	//----------------------------------------------------------------------------------------------
	// Execution of torquelimiting functionality
	//----------------------------------------------------------------------------------------------
	REGION EXECUTION_OF_TORQUELIMTING
	  // Statemachine for torquelimiting 
	  REPEAT
	    #tempStateChangeActive := FALSE;
	    CASE #statTorqueLimitingState OF
	      #NO_TORQUE_LIMITING_ACTIVE:
	        ; // Torquelimiting disable
	        // #instTorqueLimiting(Axis := #axis, V01.00.03 Dont Call MC_TORQUELIMITING if disabled
	        //                     Enable := FALSE);
	        
	      #TORQUE_LIMITING_DISABLE:
	        // Torquelimiting disable
	        #instTorqueLimiting(Axis := #axis,
	                            Enable := FALSE);
	        
	        // Check state of torque limting
	        IF (#instTorqueLimiting.Busy = FALSE)
	        THEN
	          // set next state
	          #statTorqueLimitingState := #NO_TORQUE_LIMITING_ACTIVE;
	        ELSE
	          ; // Waiting for MC_Torquelimiting is not busy
	        END_IF;
	        
	      #TORQUE_LIMTING_SELECTED:
	        // No extended homing function active
	        #instTorqueLimiting(Axis := #axis,
	                            Enable := #statExtendedCommand.%X1,
	                            Limit := #configuration.torqueLimiting.limit,
	                            Mode := #configuration.torqueLimiting.mode);
	        
	        IF (#instTorqueLimiting.Busy = FALSE) THEN
	          // Reset state
	          #statTorqueLimitingState := #NO_TORQUE_LIMITING_ACTIVE;
	        END_IF;
	        
	        (*
	        V1.00.03 Not required anymore
	      #AUTOMATIC_MODE_CHANGE:
	        // In this state the torquelimiting function is operating with Mode 1 (Fixed stop detection) until inClamping = FALSE
	        #instTorqueLimiting(Axis := #axis,
	                            Enable := TRUE,
	                            Limit := #configuration.homing.extendedModeTorqueLimit); // V01.00.03 Always use configured value
	        
	        IF (#configuration.torqueLimiting.mode = #MODE_FIXED_STOP_DETECTION)
	          OR (#instTorqueLimiting.InClamping = FALSE)
	        THEN
	          // Change state
	          #statTorqueLimitingState := #TORQUE_LIMTING_SELECTED;
	          #tempStateChangeActive := TRUE;
	        ELSE
	          ; // Wait for InClamping = FALSE
	        END_IF;
	        *)
	        
	      #FIXED_STOP_DETECTION_ACTIVE:
	        // Extended homing function active
	        #instTorqueLimiting(Axis := #axis,
	                            Enable := TRUE,
	                            Limit := #configuration.homing.extendedModeTorqueLimit, // V01.00.03 Always use configured value
	                            Mode := #MODE_FIXED_STOP_DETECTION);
	        
	        IF ((#statHomingSubState = #HOMING_IDLE) AND (#statBasicMotionState = #ACTIVE_HOMING_SELECTED))
	        THEN
	          // Fixed stop process has finished - Axis is still in clamping
	          #statTorqueLimitingState := #FIXED_STOP_DETECTION_FINISHED;
	          #tempStateChangeActive := TRUE;
	          
	        ELSIF (#statBasicMotionState <> #ACTIVE_HOMING_SELECTED)
	        THEN
	          // Error occurred - change state depending on inClamping
	          IF (#instTorqueLimiting.InClamping = TRUE)
	          THEN
	            // Axis is in clamping
	            #statTorqueLimitingState := #FIXED_STOP_DETECTION_ERROR_IN_CLAMPING;
	            #tempStateChangeActive := TRUE;
	          ELSE
	            // Axis is in not clamping
	            #statTorqueLimitingState := #FIXED_STOP_DETECTION_ERROR_NOT_IN_CLAMPING;
	            #tempStateChangeActive := TRUE;
	          END_IF;
	          
	        ELSE
	          ; // Fixed stop detection is running
	        END_IF;
	        
	      #FIXED_STOP_DETECTION_FINISHED:
	        // Homing on fixed stop process has finished
	        #instTorqueLimiting(Axis := #axis,
	                            Enable := TRUE,
	                            Limit := #configuration.homing.extendedModeTorqueLimit, // V01.00.03 Always use configured value
	                            Mode := #MODE_FIXED_STOP_DETECTION);
	        
	        IF (#instTorqueLimiting.InClamping = FALSE)
	        THEN
	          // InClamping = FALSE
	          IF (#statExtendedCommand.%X1 = TRUE) // Torquelimiting
	          THEN
	            #statTorqueLimitingState := #TORQUE_LIMTING_SELECTED;
	          ELSE
	            #statTorqueLimitingState := #TORQUE_LIMITING_DISABLE;
	          END_IF;
	          #tempStateChangeActive := TRUE;
	        ELSE
	          // InClamping = TRUE
	          IF (#statExtendedCommand.%X1 = TRUE) // Torquelimiting
	            AND (#configuration.torqueLimiting.mode = #MODE_FIXED_STOP_DETECTION)
	          THEN
	            // Change State
	            #statTorqueLimitingState := #TORQUE_LIMTING_SELECTED;
	            #tempStateChangeActive := TRUE;
	          ELSE
	            ; // Wait for inClamping = FALSE
	          END_IF;
	        END_IF;
	        
	      #FIXED_STOP_DETECTION_ERROR_IN_CLAMPING:
	        // Errorstate, torquelimiting is still active and axis not in clamping
	        #instTorqueLimiting(Axis := #axis,
	                            Enable := TRUE,
	                            Limit := #configuration.homing.extendedModeTorqueLimit, // V01.00.03 Always use configured value
	                            Mode := #MODE_FIXED_STOP_DETECTION);
	        
	        IF (#instTorqueLimiting.InClamping = FALSE)
	        THEN
	          // InClamping = FALSE -> reset torque limiting state
	          #statTorqueLimitingState := #TORQUE_LIMITING_DISABLE;
	          // Torquelimiting disable
	          #tempStateChangeActive := TRUE;
	        END_IF;
	        
	      #FIXED_STOP_DETECTION_ERROR_NOT_IN_CLAMPING:
	        // Errorstate, torquelimiting is still active and axis in clamping
	        #instTorqueLimiting(Axis := #axis,
	                            Enable := TRUE,
	                            Limit := #configuration.homing.extendedModeTorqueLimit, // V01.00.03 Always use configured value
	                            Mode := #MODE_FIXED_STOP_DETECTION);
	        
	        IF (#instTorqueLimiting.InClamping = TRUE)
	        THEN
	          // InClamping = TRUE -> change state
	          #statTorqueLimitingState := #FIXED_STOP_DETECTION_ERROR_IN_CLAMPING;
	          #tempStateChangeActive := TRUE;
	          
	        ELSIF (#statBasicMotionState <> #NO_SELECTION)
	          OR (#statSupImpMotionState <> #NO_SELECTION)
	          OR (#statPassiveHomingState <> #NO_HOMING_ACTIVE)
	        THEN
	          // New valid command is set -> reset error state
	          #statTorqueLimitingState := #TORQUE_LIMITING_DISABLE;
	          #tempStateChangeActive := TRUE;
	          
	        ELSE
	          ; // Waiting for new command or axis is getting in clamping
	        END_IF;
	      ELSE
	        // Errorhandling
	        #statStatus := #ERR_UNDEFINED_TORQUE_LIMITING_STATE;
	        #statErrorUserCleared := TRUE;
	        #diagnostics.basicMotionState := #statBasicMotionState;
	        #diagnostics.superimposedMotionState := #statSupImpMotionState;
	        #diagnostics.subfunctionStatus := 0;
	        // Set errorstate
	        #statFBState := #FB_ERROR;
	    END_CASE;
	  UNTIL (#tempStateChangeActive = FALSE)
	  END_REPEAT;
	  // Evaluate MC_Command
	  IF (#instTorqueLimiting.Error = TRUE) AND ((#statTorqueLimitingErrorOld = FALSE) OR (#statStatus = #STATUS_SUBSEQUENT_CALL)) THEN
	    // Errorhandling
	    #statStatus := #ERR_MC_TORQUELIMITING;
	    #statErrorAutoCleared := TRUE;
	    #diagnostics.basicMotionState := #statBasicMotionState;
	    #diagnostics.superimposedMotionState := #statSupImpMotionState;
	    #diagnostics.subfunctionStatus := #instTorqueLimiting.ErrorId;
	    #statFBState := #AXIS_STOP_ON_ERROR_SELECTION;
	    
	  ELSIF (#instTorqueLimiting.Error = FALSE) AND ((#statTorqueLimitingErrorOld = TRUE) AND (#statStatus = #ERR_MC_TORQUELIMITING)) THEN
	    #statStatus := #STATUS_SUBSEQUENT_CALL;
	    #statErrorAutoCleared := FALSE;
	  ELSE
	    ;
	  END_IF;
	  
	  #statTorqueLimitingErrorOld := #instTorqueLimiting.Error;
	END_REGION
	
	//----------------------------------------------------------------------------------------------
	// Selection of StopOnError / implementation of fastStop
	//----------------------------------------------------------------------------------------------
	REGION STOP_ON_ERROR
	  // Check for stopping if error occurred during execution of motion commands
	  IF (#statFBState = #AXIS_STOP_ON_ERROR_SELECTION)
	  THEN
	    #statBasicMotionState := #NO_SELECTION;
	    #statSupImpMotionState := #NO_SELECTION;
	    #statPassiveHomingState := #NO_HOMING_ACTIVE;
	    
	    IF (#configuration.generalSettings.stopOnError = TRUE)
	    THEN
	      // Read Statusword only when not already read out
	      IF (#tempStatusWord = 16#0)
	      THEN
	        #tempStatusWord := #axis.StatusWord;
	      END_IF;
	      // Evaluate error
	      IF #tempStatusWord.%X0 THEN
	        ; // Axis enabled
	        IF (#tempStatusWord.%X1 = TRUE) THEN
	          ;// TO Alarm present
	          #statFBState := #AXIS_MOTION;
	        ELSE
	          // No TO alarm present, set fastStop
	          #statBasicMotionState := #FAST_STOP_SELECTED;
	          #statFirstCycleBasicMotion := TRUE;
	          #statFBState := #AXIS_STOP_ON_ERROR_EXECUTION;
	        END_IF;
	        
	      ELSE
	        ; // Axis disabled
	        #statFBState := #AXIS_MOTION;
	      END_IF;
	      
	    ELSE
	      // Dont StopOnError
	      #statFBState := #AXIS_MOTION;
	    END_IF;
	  END_IF;
	  
	  // Implementation of fastStop
	  IF (#statBasicMotionState = #FAST_STOP_SELECTED) THEN
	    // Additional feature: Load emergency stop dynamics (TO) if no valid dynamics are configured for fastStop
	    REGION FASTSTOP SELECTED
	      // Firstcycle of command
	      IF (#statFirstCycleBasicMotion = TRUE) THEN
	        // Reset HALT command
	        #instHalt(Axis := #axis,
	                  Execute := FALSE);
	        #statFirstCycleDone := TRUE;
	        // Check dynamics for fastStop
	        // Load TO emergency Stop dynamics if value <=0 for deceleration is configured
	        IF (#configuration.fastStop.deceleration <= 0) // V1.0.2 Read TO emergencyStop deceleration only if fastStop.deceleration <= 0
	        THEN
	          // Invalid fastStop dynamics configured - read emergency stop dynamics from TO
	          #statDeceleration := #axis.DynamicDefaults.EmergencyDeceleration;
	        ELSE
	          // Valid fastStop dynamics configured
	          #statDeceleration := #configuration.fastStop.deceleration;
	        END_IF;
	        #statJerk := #configuration.fastStop.jerk; // V1.0.2 Use always configuration for jerk value
	        #statAbortAcceleration := #configuration.fastStop.abortAcceleration; // V1.0.2 Use always configuration
	      END_IF;
	      
	      // Call of MC_Command
	      #instHalt(Axis := #axis,
	                Execute := (#statBasicCommand.%X0 OR #statFirstCycleBasicMotion),
	                Deceleration := #statDeceleration,
	                AbortAcceleration := #statAbortAcceleration,
	                Jerk := #statJerk);
	      
	      // Evaluate MC_Command
	      IF (#instHalt.Busy = FALSE) AND
	        (#instHalt.Error = FALSE) AND
	        (#instHalt.Done = FALSE) AND
	        (#instHalt.CommandAborted = FALSE)
	      THEN
	        // Return to NO_SELECTION if command finished
	        #statFBState := #AXIS_MOTION;
	        #statBasicMotionState := #NO_SELECTION;
	        
	      ELSIF (#instHalt.Done = TRUE)
	      THEN
	        IF (#statFirstCycleDone = TRUE)
	        THEN
	          // Command is reset
	          IF (#instTorqueLimiting.Error = FALSE) // V1.00.03 Dont reset error is pending
	          THEN
	            // Reset status not if torquelimiting error is pending
	            #statStatus := #STATUS_SUBSEQUENT_CALL;
	            #statErrorAutoCleared := FALSE;
	          END_IF;
	          
	          #statFirstCycleDone := FALSE;
	        END_IF;
	        
	      ELSIF (#instHalt.Error = TRUE)
	      THEN
	        // Errorhandling
	        #statStatus := #ERR_MC_HALT;
	        #statErrorAutoCleared := TRUE;
	        #diagnostics := #statDiagnostics;
	        #diagnostics.basicMotionState := #statBasicMotionState;
	        #diagnostics.superimposedMotionState := #statSupImpMotionState;
	        #diagnostics.subfunctionStatus := #instHalt.ErrorId;
	        
	      ELSE
	        ; // Command selected
	      END_IF;
	      
	      // Write MC_Command outputs to internal variable
	      #statExeOfBasicMotion := 0;
	      #statExeOfBasicMotion.%X0 := #instHalt.Busy;
	      #statExeOfBasicMotion.%X1 := #instHalt.Done;
	      #statExeOfBasicMotion.%X2 := #instHalt.CommandAborted;
	      #statExeOfBasicMotion.%X3 := #instHalt.Error;
	    END_REGION
	  END_IF;
	END_REGION
	//----------------------------------------------------------------------------------------------
	// Store values and reset variables
	//----------------------------------------------------------------------------------------------
	REGION STORE_AND_RESET
	  // Reset variables to determine first cycle of a new command
	  IF (#statFirstCycleReset = TRUE) THEN
	    #statFirstCycleReset := FALSE;
	  END_IF;
	  IF (#statFirstCycleHoming = TRUE) THEN
	    #statFirstCycleHoming := FALSE;
	  END_IF;
	  #statHomingOld := #tempHoming;
	  
	  IF (#statFirstCycleBasicMotion = TRUE) THEN
	    #statFirstCycleBasicMotion := FALSE;
	  END_IF;
	  #statBasicCommandOld := #statBasicCommand;
	  
	  IF (#statFirstCycleSupImpMotion = TRUE) THEN
	    #statFirstCycleSupImpMotion := FALSE;
	  END_IF;
	  #statSupImpCommandOld := #statSupImpCommand;
	  
	  // Store last values for edge detection
	  #statEnableOld := #enable;
	  #statEnableAxisOld := #enableAxis;
	  #statExtendedCommandOld := #statExtendedCommand;
	  #statPowerErrorOld := #instPower.Error;
	END_REGION
	
	//----------------------------------------------------------------------------------------------
	// Writing outputs
	//----------------------------------------------------------------------------------------------
	REGION WRITING_OF_OUTPUTS
	  // Writing status outputs
	  #resetActive := (#statResetState = #CMD_BUSY);
	  
	  IF (#statErrorUserCleared = TRUE) THEN
	    ; // Reset variables at ErrorUserCleared
	    #statBasicMotionState := #NO_SELECTION;
	    #statExeOfBasicMotion := #NO_SELECTION;
	    #statSupImpMotionState := #NO_SELECTION;
	    #statExeOfSupImpMotionState := #NO_SELECTION;
	    #statExeOfHoming := #NO_SELECTION;
	  END_IF;
	  IF (#instPower.Status = TRUE)
	  THEN
	    // Axis enabled
	    #axisEnabled := TRUE;
	    
	  ELSIF (#instPower.Error = TRUE) AND (#instPower.Status = FALSE)
	  THEN
	    // Reset status if error occurred
	    #axisEnabled := FALSE;
	    
	  ELSIF (#instPower.Busy = FALSE)
	  THEN
	    // Reset if MC_Power is not busy
	    #axisEnabled := FALSE;
	  ELSE
	    ;
	  END_IF;
	  
	  REGION WRITING_BASICMOTION_OUTPUTS
	    // Writing Busy, Done and Aborted outputs for basic motion commands
	    IF (#statBasicMotionState > #NO_SELECTION) AND (#statBasicMotionState < #ACTIVE_HOMING_SELECTED)
	    THEN
	      #commandBusy := #statExeOfBasicMotion.%X0;
	      #commandDone := #statExeOfBasicMotion.%X1;
	      #commandAborted := #statExeOfBasicMotion.%X2;
	      #inVelocity := #statExeOfBasicMotion.%X4;
	    ELSE
	      #commandBusy := FALSE;
	      #commandDone := FALSE;
	      #commandAborted := FALSE;
	      #inVelocity := FALSE;
	    END_IF;
	    
	    // Writing outputs up to LAxisCtrl_SpeedAxis
	    IF (#statTorqueLimitingState = #TORQUE_LIMTING_SELECTED)
	      // OR (#statTorqueLimitingState = #AUTOMATIC_MODE_CHANGE) V1.0.3 TorqueLimtinig = TRUE, only when respective value used 
	    THEN
	      #torqueLimitingSelected := TRUE;
	    ELSE
	      #torqueLimitingSelected := FALSE;
	    END_IF;
	    
	    #inLimitation := #instTorqueLimiting.InLimitation;
	    #fastStopSelected := #statBasicMotionState.%X0;
	    #stopSelected := #statBasicMotionState.%X1;
	    #jogSelected := #statBasicMotionState.%X2 OR #statBasicMotionState.%X3;
	    #moveVelocitySelected := #statBasicMotionState.%X4;
	    // Writing outputs up to LAxisCtrl_PosAxis
	    #inClamping := #instTorqueLimiting.InClamping;
	    #posRelativeSelected := #statBasicMotionState.%X5;
	    #posAbsoluteSelected := #statBasicMotionState.%X6;
	  END_REGION
	  REGION WRITING_HOMING_OUTPUTS
	    // Writing Busy, Done and Aborted outputs for homing
	    IF (#statPassiveHomingState = #STANDARD_HOMING)
	    THEN
	      #homingSelected := TRUE;
	      #homingCommandBusy := #statExeOfHoming.%X0;
	      #homingCommandDone := #statExeOfHoming.%X1;
	      #homingCommandAborted := #statExeOfHoming.%X2;
	    ELSE
	      IF (#statBasicMotionState = #ACTIVE_HOMING_SELECTED)
	      THEN
	        #homingSelected := TRUE;
	        #homingCommandBusy := #statExeOfBasicMotion.%X0;
	        #homingCommandDone := #statExeOfBasicMotion.%X1;
	        #homingCommandAborted := #statExeOfBasicMotion.%X2;
	      ELSE
	        #homingSelected := FALSE;
	        #homingCommandBusy := FALSE;
	        #homingCommandDone := FALSE;
	        #homingCommandAborted := FALSE;
	      END_IF;
	    END_IF;
	  END_REGION
	  REGION WRITING_SUPERIMPOSED_OUTPUTS
	    // Writing outputs for superimposed motion commands
	    IF (#statSupImpMotionState <> #NO_SELECTION)
	    THEN
	      #superimposedBusy := #statExeOfSupImpMotionState.%X0;
	      #superimposedDone := #statExeOfSupImpMotionState.%X1;
	      #superimposedAborted := #statExeOfSupImpMotionState.%X2;
	    ELSE
	      #superimposedBusy := FALSE;
	      #superimposedDone := FALSE;
	      #superimposedAborted := FALSE;
	    END_IF;
	    #posSuperimposedSelected := #statSupImpMotionState.%X0;
	  END_REGION
	END_REGION
	
	//----------------------------------------------------------------------------------------------
	// Error handling 
	//----------------------------------------------------------------------------------------------
	REGION ERROR_HANDLING
	  IF #statErrorUserCleared THEN
	    #valid := FALSE;
	    #busy := TRUE;
	    #error := TRUE;
	    #status := #statStatus;
	    #diagnostics.status := #statStatus;
	    
	  ELSIF #statErrorAutoCleared THEN
	    #valid := FALSE;
	    #busy := TRUE;
	    #error := TRUE;
	    #status := #statStatus;
	    #diagnostics.status := #statStatus;
	    
	  ELSE
	    // Process normal output values
	    #valid := TRUE;
	    #error := FALSE;
	    #status := #statStatus;
	  END_IF;
	END_REGION
END_FUNCTION_BLOCK

FUNCTION_BLOCK "FB_Axis"   // FB30140, LAD
{ S7_Optimized_Access := 'TRUE' }
// stored: AutoNumber false, MemoryReserve 100, SetENOAutomatically false
   VAR_INPUT
      TO_PosAxis : TO_PositioningAxis;
      I_bMan_Enable : Bool;
      I_iHomeMode : Int;
      I_iHomePos : LReal;
   END_VAR
   VAR_IN_OUT
      Ds_Axis : "sAxis";
   END_VAR
   VAR
      instAxis01 { ExternalAccessible := 'False'; ExternalVisible := 'False'; ExternalWritable := 'False'} : "LAxisCtrl_PosAxis";
      instShearAxisStatus { S7_SetPoint := 'True'} : "LAxisCtrl_GetAxisStatusWord";
      RT_Reset { S7_SetPoint := 'True'} : R_TRIG;
      RT_PB { ExternalAccessible := 'False'; ExternalVisible := 'False'; ExternalWritable := 'False'} : Array[0..19] of R_TRIG;   // Störungen / Alarms
      FT_PB { ExternalAccessible := 'False'; ExternalVisible := 'False'; ExternalWritable := 'False'; S7_SetPoint := 'True'} : Array[0..19] of F_TRIG;   // Störungen unterdrücken, Belegung identisch mit "Alarm" / Hide Alarms, identical with "Alarm"
      TON_PB { ExternalAccessible := 'False'; ExternalVisible := 'False'; ExternalWritable := 'False'} : Array[0..19] of TON_TIME;   // Fallende Flanke / Falling edge
      TOF_PB { ExternalAccessible := 'False'; ExternalVisible := 'False'; ExternalWritable := 'False'} : Array[0..19] of TOF_TIME;   // Negativer Impuls / Negative pulse
      i { S7_SetPoint := 'True'} : Int;
      temp_cmd_bEnableAxis { ExternalAccessible := 'False'; ExternalVisible := 'False'; ExternalWritable := 'False'} : Bool;
      temp_cmd_bresetAxis { ExternalAccessible := 'False'; ExternalVisible := 'False'; ExternalWritable := 'False'} : Bool;
      temp_cmd_bjogForward { ExternalAccessible := 'False'; ExternalVisible := 'False'; ExternalWritable := 'False'} : Bool;
      temp_cmd_bjogBackward { ExternalAccessible := 'False'; ExternalVisible := 'False'; ExternalWritable := 'False'} : Bool;
      temp_cmd_bmoveVelocity { ExternalAccessible := 'False'; ExternalVisible := 'False'; ExternalWritable := 'False'} : Bool;
      temp_cmd_bstop { ExternalAccessible := 'False'; ExternalVisible := 'False'; ExternalWritable := 'False'} : Bool;
      temp_cmd_bfastStop { ExternalAccessible := 'False'; ExternalVisible := 'False'; ExternalWritable := 'False'} : Bool;
      temp_cmd_bhoming { ExternalAccessible := 'False'; ExternalVisible := 'False'; ExternalWritable := 'False'} : Bool;
      temp_cmd_bGoToPos { ExternalAccessible := 'False'; ExternalVisible := 'False'; ExternalWritable := 'False'} : Array[0..16] of Bool;
      temp_cmd_iGoToPos : Word;
      temp_cmd_bCallAbsPos : Bool;
      temp_cmd_bRelPos : Bool;
      temp_Para_rJog_Speed { ExternalAccessible := 'False'; ExternalVisible := 'False'; ExternalWritable := 'False'} : LReal;
      temp_cmd_bGoToPosAll { ExternalAccessible := 'False'; ExternalVisible := 'False'; ExternalWritable := 'False'} : Bool;
      temp_configuration { ExternalAccessible := 'False'; ExternalVisible := 'False'; ExternalWritable := 'False'} : "LAxisCtrl_typeAxisConfig";   // Diagnostics structure
      temp_Status { ExternalAccessible := 'False'; ExternalVisible := 'False'; ExternalWritable := 'False'} : Word;
      tempAxisEnabled { ExternalAccessible := 'False'; ExternalVisible := 'False'; ExternalWritable := 'False'} : Bool;
      temp_CommandBusy { ExternalAccessible := 'False'; ExternalVisible := 'False'; ExternalWritable := 'False'} : Bool;
      temp_CommandDone { ExternalAccessible := 'False'; ExternalVisible := 'False'; ExternalWritable := 'False'} : Bool;
      temp_CommandAborted { ExternalAccessible := 'False'; ExternalVisible := 'False'; ExternalWritable := 'False'} : Bool;
      temp_InVelocity { ExternalAccessible := 'False'; ExternalVisible := 'False'; ExternalWritable := 'False'} : Bool;
      temp_jogSelected { ExternalAccessible := 'False'; ExternalVisible := 'False'; ExternalWritable := 'False'} : Bool;
      tempPosAbsoluteSelected { ExternalAccessible := 'False'; ExternalVisible := 'False'; ExternalWritable := 'False'} : Bool;
      temp_diagnostics { ExternalAccessible := 'False'; ExternalVisible := 'False'; ExternalWritable := 'False'} : "LAxisCtrl_typeDiagnostics";
      temp_stop_Dec { ExternalAccessible := 'False'; ExternalVisible := 'False'; ExternalWritable := 'False'} : LReal;
      temp_faststop_Dec { ExternalAccessible := 'False'; ExternalVisible := 'False'; ExternalWritable := 'False'} : LReal;
      temp_iFBStatus : Word;
      temp_iMCStatus : Word;
      old_iFBStatus : Word;
      old_iMCStatus : Word;
   END_VAR
BEGIN

REGION Network 1
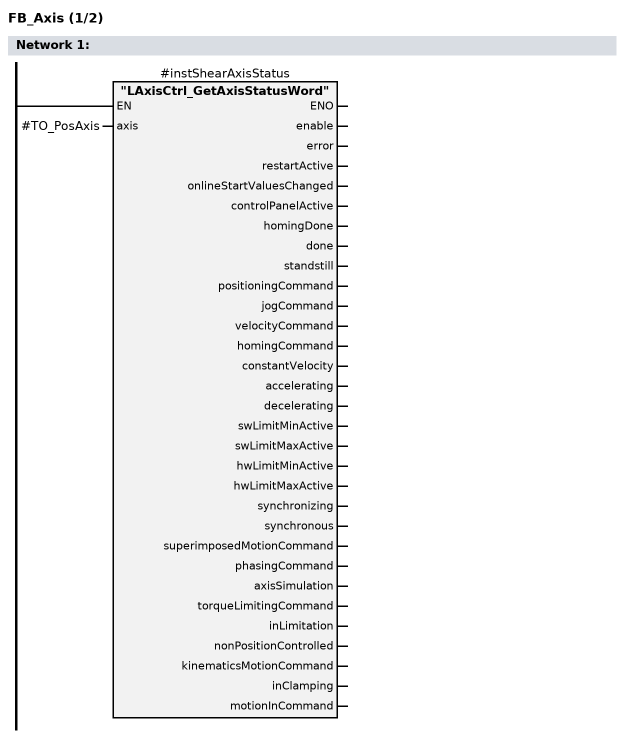
   RUNG wire#powerrail
      #instShearAxisStatus(axis := #TO_PosAxis, enable =>, error =>, restartActive =>, onlineStartValuesChanged =>, controlPanelActive =>, homingDone =>, done =>, standstill =>, positioningCommand =>, jogCommand =>, velocityCommand =>, homingCommand =>, constantVelocity =>, accelerating =>, decelerating =>, swLimitMinActive =>, swLimitMaxActive =>, hwLimitMinActive =>, hwLimitMaxActive =>, synchronizing =>, synchronous =>, superimposedMotionCommand =>, phasingCommand =>, axisSimulation =>, torqueLimitingCommand =>, inLimitation =>, nonPositionControlled =>, kinematicsMotionCommand =>, inClamping =>, motionInCommand =>)
   END_RUNG
   // the same network as SCL:
   #instShearAxisStatus(axis := #TO_PosAxis);   // "LAxisCtrl_GetAxisStatusWord"
END_REGION

REGION Network 2: LAxisCtrl
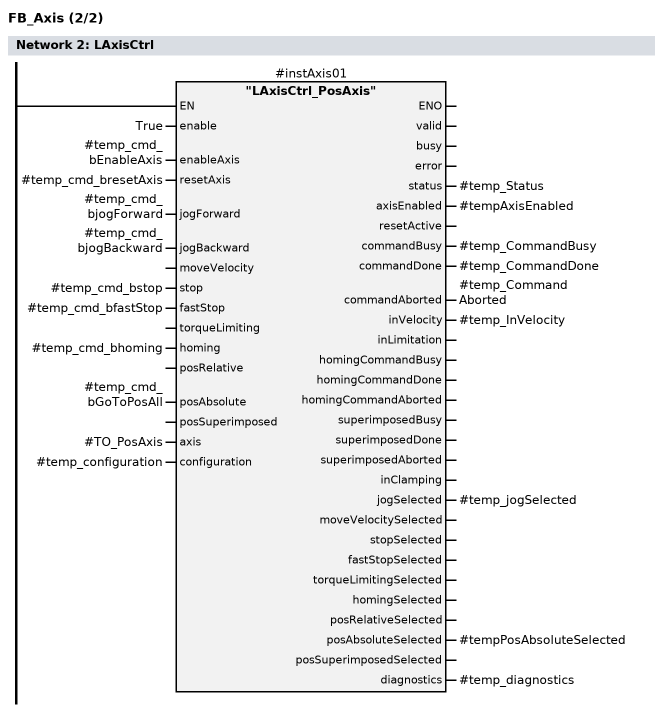
   RUNG wire#powerrail
      #instAxis01(enable := True, enableAxis := #temp_cmd_bEnableAxis, resetAxis := #temp_cmd_bresetAxis, jogForward := #temp_cmd_bjogForward, jogBackward := #temp_cmd_bjogBackward, moveVelocity :=, stop := #temp_cmd_bstop, fastStop := #temp_cmd_bfastStop, torqueLimiting :=, homing := #temp_cmd_bhoming, posRelative :=, posAbsolute := #temp_cmd_bGoToPosAll, posSuperimposed :=, axis := #TO_PosAxis, configuration := #temp_configuration, valid =>, busy =>, error =>, status => #temp_Status, axisEnabled => #tempAxisEnabled, resetActive =>, commandBusy => #temp_CommandBusy, commandDone => #temp_CommandDone, commandAborted => #temp_CommandAborted, inVelocity => #temp_InVelocity, inLimitation =>, homingCommandBusy =>, homingCommandDone =>, homingCommandAborted =>, superimposedBusy =>, superimposedDone =>, superimposedAborted =>, inClamping =>, jogSelected => #temp_jogSelected, moveVelocitySelected =>, stopSelected =>, fastStopSelected =>, torqueLimitingSelected =>, homingSelected =>, posRelativeSelected =>, posAbsoluteSelected => #tempPosAbsoluteSelected, posSuperimposedSelected =>, diagnostics => #temp_diagnostics)
   END_RUNG
   // the same network as SCL:
   #instAxis01(enable := True,   // "LAxisCtrl_PosAxis"
               enableAxis := #temp_cmd_bEnableAxis,
               resetAxis := #temp_cmd_bresetAxis,
               jogForward := #temp_cmd_bjogForward,
               jogBackward := #temp_cmd_bjogBackward,
               stop := #temp_cmd_bstop,
               fastStop := #temp_cmd_bfastStop,
               homing := #temp_cmd_bhoming,
               posAbsolute := #temp_cmd_bGoToPosAll,
               axis := #TO_PosAxis,
               configuration := #temp_configuration,
               status => #temp_Status,
               axisEnabled => #tempAxisEnabled,
               commandBusy => #temp_CommandBusy,
               commandDone => #temp_CommandDone,
               commandAborted => #temp_CommandAborted,
               inVelocity => #temp_InVelocity,
               jogSelected => #temp_jogSelected,
               posAbsoluteSelected => #tempPosAbsoluteSelected,
               diagnostics => #temp_diagnostics);
END_REGION

REGION Network 3 (SCL): input
   #temp_cmd_bEnableAxis  := #Ds_Axis.I_CMD.bEnableAxis OR (#Ds_Axis.I_HMI.bEnableAxis AND #I_bMan_Enable);
   #temp_cmd_bresetAxis   := #Ds_Axis.I_CMD.bResetAxis;
   #temp_cmd_bjogForward  := #Ds_Axis.I_InLock.bjogForward AND (#Ds_Axis.I_CMD.bjogForward OR (#Ds_Axis.I_HMI.bjogForward AND #I_bMan_Enable)) ;
   #temp_cmd_bjogBackward := #Ds_Axis.I_InLock.bjogBackward AND (#Ds_Axis.I_CMD.bjogBackward OR (#Ds_Axis.I_HMI.bjogBackward AND #I_bMan_Enable)) ;
   #temp_cmd_bstop        := #Ds_Axis.I_CMD.bstop OR (#Ds_Axis.I_HMI.bstop AND #I_bMan_Enable);
   #temp_cmd_bfastStop    := #Ds_Axis.I_CMD.bfastStop;
   #temp_cmd_bhoming      := #Ds_Axis.I_InLock.bHoming AND (#Ds_Axis.I_CMD.bHoming OR #Ds_Axis.I_HMI.bHoming) ;
END_REGION

REGION Network 4 (SCL): Configuration
   #Ds_Axis.I_Para.rJog_Speed[0] := 10.0;
   #Ds_Axis.I_Para.rMV_Speed[0] := 100.0;
   #Ds_Axis.I_Para.rStop_Dec[0] := 20.0;
   #Ds_Axis.I_Para.rEStop_Dec[0] := 50.0;

   #Ds_Axis.I_Para.rJog_Speed[1] := 100.0 * #Ds_Axis.I_Para.rJog_Speed[0];
   #Ds_Axis.I_Para.rJog_Speed[2] := 100.0 * #Ds_Axis.I_Para.rJog_Speed[0];
   #Ds_Axis.I_Para.rMV_Speed[1] := 100.0 * #Ds_Axis.I_Para.rMV_Speed[0];
   #Ds_Axis.I_Para.rMV_Speed[2] := 100.0 * #Ds_Axis.I_Para.rMV_Speed[0];
   #Ds_Axis.I_Para.rStop_Dec[1] := 100.0 * #Ds_Axis.I_Para.rStop_Dec[0];
   #Ds_Axis.I_Para.rEStop_Dec[1] := 100.0 * #Ds_Axis.I_Para.rEStop_Dec[0];

   IF #temp_configuration.jog.velocity <> #Ds_Axis.I_Para.rJog_Speed[0] OR
       #temp_configuration.jog.acceleration <> #Ds_Axis.I_Para.rJog_Speed[1] OR
       #temp_configuration.jog.deceleration <> #Ds_Axis.I_Para.rJog_Speed[2] OR
       #temp_configuration.moveVelocity.acceleration <> #Ds_Axis.I_Para.rMV_Speed[0] OR
       #temp_configuration.moveVelocity.deceleration <> #Ds_Axis.I_Para.rMV_Speed[1] OR
       #temp_configuration.moveVelocity.acceleration <> #Ds_Axis.I_Para.rMV_Speed[2] OR
       #temp_configuration.stop.deceleration <> #Ds_Axis.I_Para.rStop_Dec[0] OR
       #temp_configuration.stop.jerk <> #Ds_Axis.I_Para.rStop_Dec[1] OR
       #temp_configuration.fastStop.deceleration <> #Ds_Axis.I_Para.rEStop_Dec[0] OR
       #temp_configuration.fastStop.jerk <> #Ds_Axis.I_Para.rEStop_Dec[1]
   THEN
       // Jog
       #temp_configuration.jog.velocity := #Ds_Axis.I_Para.rJog_Speed[0];
       #temp_configuration.jog.acceleration := #Ds_Axis.I_Para.rJog_Speed[1];
       #temp_configuration.jog.deceleration := #Ds_Axis.I_Para.rJog_Speed[2];
       // Move
       #temp_configuration.moveVelocity.velocity := #Ds_Axis.I_Para.rMV_Speed[0];
       #temp_configuration.moveVelocity.acceleration := #Ds_Axis.I_Para.rMV_Speed[1];
       #temp_configuration.moveVelocity.deceleration := #Ds_Axis.I_Para.rMV_Speed[2];
       // Stop   
       #temp_configuration.stop.deceleration := #Ds_Axis.I_Para.rStop_Dec[0];
       #temp_configuration.stop.jerk := #Ds_Axis.I_Para.rStop_Dec[1];
       //faststoo
       #temp_configuration.fastStop.deceleration := #Ds_Axis.I_Para.rEStop_Dec[0];
       #temp_configuration.fastStop.jerk := #Ds_Axis.I_Para.rEStop_Dec[1];
   END_IF;

   // Homing
   #temp_configuration.homing.mode := #I_iHomeMode;//I_iHomeMode
   #temp_configuration.homing.position := #I_iHomePos;//I_iHomePos

   //AbsPos
   //#temp_cmd_bGoToPosAll := #Ds_Axis.I_CMD.bCallAbsPos AND #Ds_Axis.I_InLock.bGoToPos[1];//"dStruct_Axis".gs_Axis[0].I_CMD.bCallAbsPos
   #temp_cmd_bGoToPosAll := "dStruct_Axis".gs_Axis[0].I_HMI.bCallAbsPos AND #Ds_Axis.I_InLock.bGoToPos[1];
   //#temp_posAbsolute :=
   //#Ds_Axis.I_bGoToPos[0] OR #Ds_Axis.I_bGoToPos[1] OR #Ds_Axis.I_bGoToPos[2] OR #Ds_Axis.I_bGoToPos[3] OR
   //#Ds_Axis.I_bGoToPos[4] OR #Ds_Axis.I_bGoToPos[5] OR #Ds_Axis.I_bGoToPos[6] OR #Ds_Axis.I_bGoToPos[7] OR
   //#Ds_Axis.I_bGoToPos[8] OR #Ds_Axis.I_bGoToPos[9] OR #Ds_Axis.I_bGoToPos[10] OR #Ds_Axis.I_bGoToPos[11] OR
   //#Ds_Axis.I_bGoToPos[12] OR #Ds_Axis.I_bGoToPos[13] OR #Ds_Axis.I_bGoToPos[14] OR #Ds_Axis.I_bGoToPos[15];

   #temp_configuration.posAbsolute.position := "dStruct_Axis".gs_Axis[0].I_Para.rPos_Abs[0];//#Ds_Axis.I_Para.rPos_Abs[0];
   #temp_configuration.posAbsolute.velocity := "dStruct_Axis".gs_Axis[0].I_Para.rSpeed_Abs[0];//#Ds_Axis.I_Para.rSpeed_Abs[0];
   #temp_configuration.posAbsolute.direction := 3;

   #temp_configuration.posAbsolute.acceleration := #temp_configuration.posAbsolute.velocity * 10.0;//#Ds_Axis.Para.I_iAcc_Set;
   #temp_configuration.posAbsolute.deceleration := #temp_configuration.posAbsolute.velocity * 10.0;//#Ds_Axis.Para.I_iDec_Set;
   #temp_configuration.posAbsolute.jerk := #temp_configuration.posAbsolute.velocity * 100.0;//#Ds_Axis.Para.I_iJerk_Set;

   (*
   FOR #i := 0 TO 15 DO
   //    #RT_PB[#i](CLK := #Ds_Axis.I_bGoToPos[#i]);
       #RT_PB[#i](CLK := #Ds_Axis.CMD.I_bCallAbsPos);

       IF #RT_PB[#i].Q THEN
           #temp_configuration.posAbsolute.position := #Ds_Axis.Para.I_rPos_Abs[0];
           #temp_configuration.posAbsolute.velocity := #Ds_Axis.Para.I_rSpeed_Abs[0];
           #temp_configuration.posAbsolute.direction := 3;//temp_posAbsolute_direction

           #temp_configuration.posAbsolute.acceleration := #Ds_Axis.Para.I_iAcc_Set;
           #temp_configuration.posAbsolute.deceleration := #Ds_Axis.Para.I_iDec_Set;
           #temp_configuration.posAbsolute.jerk := #Ds_Axis.Para.I_iJerk_Set;

       END_IF;
   END_FOR;
   *)
END_REGION

REGION Network 5 (SCL): output
   #Ds_Axis.O_Status.bAxisEnabled := #tempAxisEnabled;
   #Ds_Axis.O_Status.bjogForward := #temp_cmd_bjogForward;//AND #temp_jogSelected ;
   #Ds_Axis.O_Status.bjogBackward := #temp_cmd_bjogBackward;//AND #temp_jogSelected;
   #Ds_Axis.O_Status.bHomed := #TO_PosAxis.StatusWord.%X5;
   #Ds_Axis.O_Status.bAxisError := #TO_PosAxis.StatusWord.%X1;
   #Ds_Axis.O_Status.rActPos := #TO_PosAxis.ActualPosition;
   #Ds_Axis.O_Status.rActSpeed := #TO_PosAxis.ActualVelocity;
   #Ds_Axis.O_Status.iAxisFaultNum := #TO_PosAxis.ErrorDetail.Number;
   //#Ds_Axis.O_DriveFaultNum
   //#Ds_Axis.O_Status.iFBStatus := #temp_diagnostics.status;
   //#Ds_Axis.O_Status.iMCStatus := #temp_diagnostics.subfunctionStatus;
   //#Ds_Axis.O_Torque
   //#Ds_Axis.oAxisName  := 


   #Ds_Axis.O_Status.bAtPos[0] := "FC_bNearIn"(rAct := #Ds_Axis.O_Status.rActPos, rTgt := #Ds_Axis.I_Para.rPos_Abs[0], rDelta := 1.0, bModule := 0, rModulo := 0);


   //#Ds_Axis.O_bPosDone
   //#Ds_Axis.O_bPosing
   //#tempPosAbsoluteSelected
END_REGION

REGION Network 6 (SCL): Reset
   #RT_Reset(CLK := #temp_cmd_bresetAxis);
   IF #RT_Reset.Q THEN
       #Ds_Axis.O_Status.iFBStatus := 16#00;
       #Ds_Axis.O_Status.iMCStatus := 16#00;
   END_IF;

   #temp_iFBStatus := #temp_diagnostics.status;
   IF #temp_iFBStatus <> #old_iFBStatus THEN
       #Ds_Axis.O_Status.iFBStatus := #temp_diagnostics.status;
       #old_iFBStatus := #temp_iFBStatus;
   END_IF;
   #temp_iMCStatus := #temp_diagnostics.subfunctionStatus;
   IF #temp_iMCStatus <> #old_iMCStatus THEN
       #Ds_Axis.O_Status.iFBStatus := #temp_diagnostics.subfunctionStatus;
       #old_iMCStatus := #temp_iMCStatus;
   END_IF;
END_REGION
END_FUNCTION_BLOCK

FUNCTION_BLOCK "COLLECTIVE_OR_SIGNAL_FB"   // FB41, LAD
TITLE = COLLECTIVE_OR_SIGNAL_FB / COLLECTIVE_OR_SIGNAL_FC
{ S7_Optimized_Access := 'TRUE' }
AUTHOR : Tesla
FAMILY : Alarm_PD
VERSION : 1.0
// Der Baustein verodert 16 Eingangssignale (SIGNAL_1…SIGNAL_16) zu einem Ausgangssignal (COLLECTIVE_SIGNAL).
// Verwendungszweck (Beispiel): Zur Bildung eines Sammelsignals (z.B. für eine Sammelfehler-Leuchte für "Alarme", "Warnungen", "Infos") aus den Kategorie-Informationen der ProDiag-IDBs.
// The block converts 16 input signals (SIGNAL_1 ... SIGNAL_16) into an output signal (COLLECTIVE_SIGNAL), with OR-function.
// Purpose (example): To form a collection signal (e.g., a collective error light for "alarms," "warnings," "info") from the category information of the ProDiag IDBs.
// block converts 16 输入 信号 (SIGNAL_1 ... SIGNAL_16) into an 输出 信号 (COLLECTIVE_SIGNAL), 有 或者-功能.
// Purpose (例子): 到 form a collection 信号 (e.g., a collective 错误 light 给 "警报," "warnings," "信息") 从  类别 信息 of  ProDiag IDBs.
// stored: MemoryReserve 100, SetENOAutomatically false
   VAR_INPUT
      SIGNAL_1 { ExternalAccessible := 'False'; ExternalVisible := 'False'; ExternalWritable := 'False'} : Bool;   // Eingangs-Signal (Bool) / Input signal (Bool) / 输入 信号 (Bool)
      SIGNAL_2 { ExternalAccessible := 'False'; ExternalVisible := 'False'; ExternalWritable := 'False'} : Bool;   // Eingangs-Signal (Bool) / Input signal (Bool) / 输入 信号 (Bool)
      SIGNAL_3 { ExternalAccessible := 'False'; ExternalVisible := 'False'; ExternalWritable := 'False'} : Bool;   // Eingangs-Signal (Bool) / Input signal (Bool) / 输入 信号 (Bool)
      SIGNAL_4 { ExternalAccessible := 'False'; ExternalVisible := 'False'; ExternalWritable := 'False'} : Bool;   // Eingangs-Signal (Bool) / Input signal (Bool) / 输入 信号 (Bool)
      SIGNAL_5 { ExternalAccessible := 'False'; ExternalVisible := 'False'; ExternalWritable := 'False'} : Bool;   // Eingangs-Signal (Bool) / Input signal (Bool) / 输入 信号 (Bool)
      SIGNAL_6 { ExternalAccessible := 'False'; ExternalVisible := 'False'; ExternalWritable := 'False'} : Bool;   // Eingangs-Signal (Bool) / Input signal (Bool) / 输入 信号 (Bool)
      SIGNAL_7 { ExternalAccessible := 'False'; ExternalVisible := 'False'; ExternalWritable := 'False'} : Bool;   // Eingangs-Signal (Bool) / Input signal (Bool) / 输入 信号 (Bool)
      SIGNAL_8 { ExternalAccessible := 'False'; ExternalVisible := 'False'; ExternalWritable := 'False'} : Bool;   // Eingangs-Signal (Bool) / Input signal (Bool) / 输入 信号 (Bool)
      SIGNAL_9 { ExternalAccessible := 'False'; ExternalVisible := 'False'; ExternalWritable := 'False'} : Bool;   // Eingangs-Signal (Bool) / Input signal (Bool) / 输入 信号 (Bool)
      SIGNAL_10 { ExternalAccessible := 'False'; ExternalVisible := 'False'; ExternalWritable := 'False'} : Bool;   // Eingangs-Signal (Bool) / Input signal (Bool) / 输入 信号 (Bool)
      SIGNAL_11 { ExternalAccessible := 'False'; ExternalVisible := 'False'; ExternalWritable := 'False'} : Bool;   // Eingangs-Signal (Bool) / Input signal (Bool) / 输入 信号 (Bool)
      SIGNAL_12 { ExternalAccessible := 'False'; ExternalVisible := 'False'; ExternalWritable := 'False'} : Bool;   // Eingangs-Signal (Bool) / Input signal (Bool) / 输入 信号 (Bool)
      SIGNAL_13 { ExternalAccessible := 'False'; ExternalVisible := 'False'; ExternalWritable := 'False'} : Bool;   // Eingangs-Signal (Bool) / Input signal (Bool) / 输入 信号 (Bool)
      SIGNAL_14 { ExternalAccessible := 'False'; ExternalVisible := 'False'; ExternalWritable := 'False'} : Bool;   // Eingangs-Signal (Bool) / Input signal (Bool) / 输入 信号 (Bool)
      SIGNAL_15 { ExternalAccessible := 'False'; ExternalVisible := 'False'; ExternalWritable := 'False'} : Bool;   // Eingangs-Signal (Bool) / Input signal (Bool) / 输入 信号 (Bool)
      SIGNAL_16 { ExternalAccessible := 'False'; ExternalVisible := 'False'; ExternalWritable := 'False'} : Bool;   // Eingangs-Signal (Bool) / Input signal (Bool) / 输入 信号 (Bool)
   END_VAR
   VAR_OUTPUT
      COLLECTIVE_SIGNAL : Bool;   // Ausgangs-Summensignal (Bool) / Output Collective signal (Bool) / 输出 Collective 信号 (Bool)
   END_VAR
BEGIN

REGION Network 1: Ausgangs-Summensignal (Bool) / Output Collective signal (Bool) / 输出 Collective 信号 (Bool)
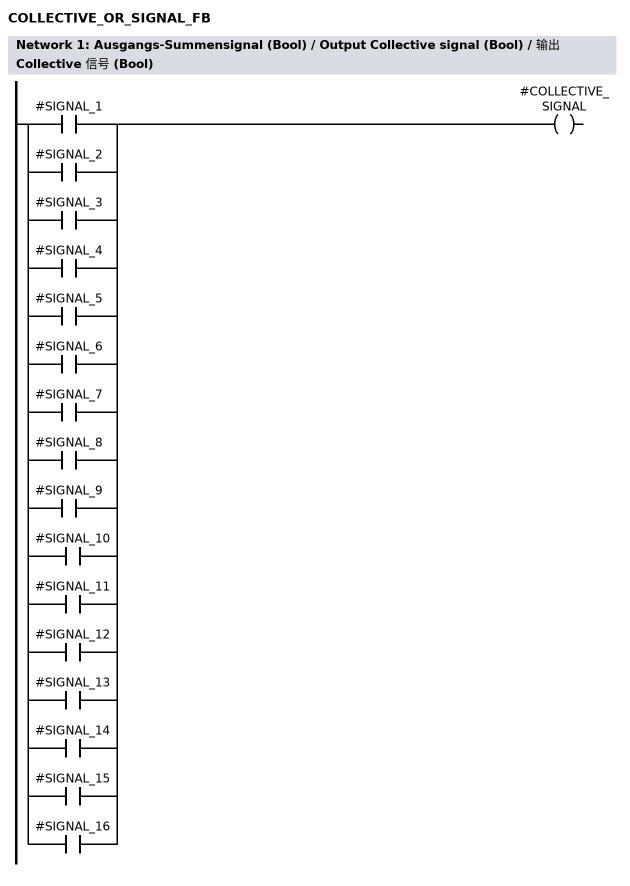
   RUNG wire#powerrail
      Contact( #SIGNAL_1 )
      wire#w1
      Coil( #COLLECTIVE_SIGNAL )
   END_RUNG
   RUNG wire#powerrail
      Contact( #SIGNAL_2 )
   END_RUNG wire#w1
   RUNG wire#powerrail
      Contact( #SIGNAL_3 )
   END_RUNG wire#w1
   RUNG wire#powerrail
      Contact( #SIGNAL_4 )
   END_RUNG wire#w1
   RUNG wire#powerrail
      Contact( #SIGNAL_5 )
   END_RUNG wire#w1
   RUNG wire#powerrail
      Contact( #SIGNAL_6 )
   END_RUNG wire#w1
   RUNG wire#powerrail
      Contact( #SIGNAL_7 )
   END_RUNG wire#w1
   RUNG wire#powerrail
      Contact( #SIGNAL_8 )
   END_RUNG wire#w1
   RUNG wire#powerrail
      Contact( #SIGNAL_9 )
   END_RUNG wire#w1
   RUNG wire#powerrail
      Contact( #SIGNAL_10 )
   END_RUNG wire#w1
   RUNG wire#powerrail
      Contact( #SIGNAL_11 )
   END_RUNG wire#w1
   RUNG wire#powerrail
      Contact( #SIGNAL_12 )
   END_RUNG wire#w1
   RUNG wire#powerrail
      Contact( #SIGNAL_13 )
   END_RUNG wire#w1
   RUNG wire#powerrail
      Contact( #SIGNAL_14 )
   END_RUNG wire#w1
   RUNG wire#powerrail
      Contact( #SIGNAL_15 )
   END_RUNG wire#w1
   RUNG wire#powerrail
      Contact( #SIGNAL_16 )
   END_RUNG wire#w1
   // the same network as SCL:
   #COLLECTIVE_SIGNAL := #SIGNAL_1 OR #SIGNAL_2 OR #SIGNAL_3 OR #SIGNAL_4 OR #SIGNAL_5 OR #SIGNAL_6 OR #SIGNAL_7 OR #SIGNAL_8 OR #SIGNAL_9 OR #SIGNAL_10 OR #SIGNAL_11 OR #SIGNAL_12 OR #SIGNAL_13 OR #SIGNAL_14 OR #SIGNAL_15 OR #SIGNAL_16;
END_REGION

NETWORK
TITLE = Baustein-Ende / End of block / 结束 of block
// ENO immer "1" setzen mit SET & SAVE / ENO always set to "1" with SET & SAVE / ENO 总是 设置 到 "1" 有 设置 & 保存
      SET;
      SAVE;
END_FUNCTION_BLOCK

FUNCTION "OneMES_HMI_Control" : Void   // FC20230, LAD
{ S7_Optimized_Access := 'TRUE' }
// stored: AutoNumber false, SetENOAutomatically false
   VAR_INPUT
      iManualMode : Bool;
      iOP_Sum : SInt;
   END_VAR
   VAR_IN_OUT
      ioHMI : "UDT_OneMES_HMI_Control";
      ioOP : Array[1.."OP_Sum"] of "UDT_MESControl";
      ioPluse : Bool;
   END_VAR
   VAR_TEMP   // added for the SCL form of the ladder/FBD networks
      _w1 : Bool;
   END_VAR
BEGIN

REGION Network 1: OP Limit
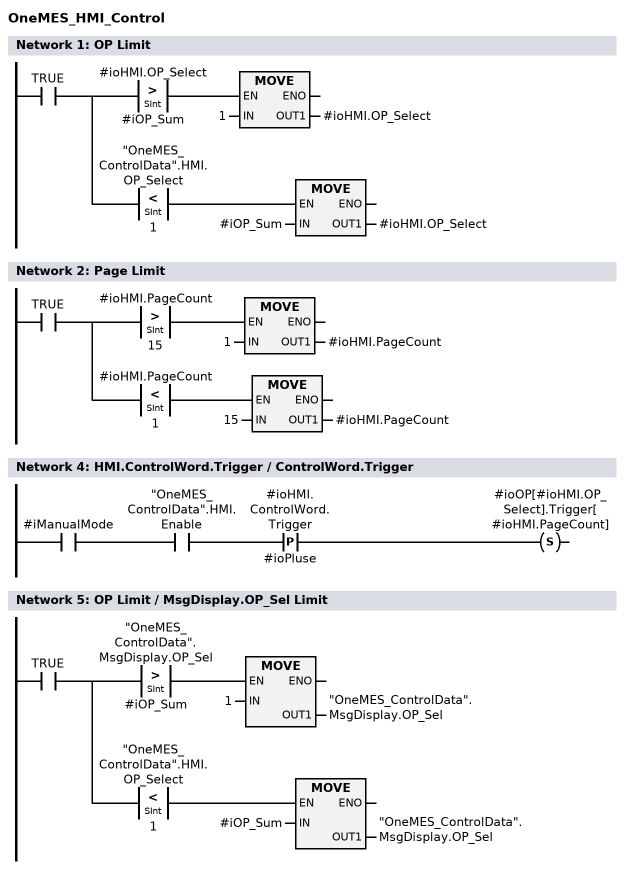
   RUNG wire#powerrail
      Contact( TRUE )
      wire#w1
      { S7_Templates := "SrcType := SInt" } GT_Contact(in1 := #ioHMI.OP_Select, in2 := #iOP_Sum)
      Move(in := 1, out1 => #ioHMI.OP_Select)
   END_RUNG
   RUNG wire#w1
      { S7_Templates := "SrcType := SInt" } LT_Contact(in1 := "OneMES_ControlData".HMI.OP_Select, in2 := 1)
      Move(in := #iOP_Sum, out1 => #ioHMI.OP_Select)
   END_RUNG
   // the same network as SCL:
   IF TRUE AND (#ioHMI.OP_Select > #iOP_Sum) THEN #ioHMI.OP_Select := 1; END_IF;
   IF TRUE AND ("OneMES_ControlData".HMI.OP_Select < 1) THEN #ioHMI.OP_Select := #iOP_Sum; END_IF;
END_REGION

REGION Network 2: Page Limit
   RUNG wire#powerrail
      Contact( TRUE )
      wire#w1
      { S7_Templates := "SrcType := SInt" } GT_Contact(in1 := #ioHMI.PageCount, in2 := 15)
      Move(in := 1, out1 => #ioHMI.PageCount)
   END_RUNG
   RUNG wire#w1
      { S7_Templates := "SrcType := SInt" } LT_Contact(in1 := #ioHMI.PageCount, in2 := 1)
      Move(in := 15, out1 => #ioHMI.PageCount)
   END_RUNG
   // the same network as SCL:
   IF TRUE AND (#ioHMI.PageCount > 15) THEN #ioHMI.PageCount := 1; END_IF;
   IF TRUE AND (#ioHMI.PageCount < 1) THEN #ioHMI.PageCount := 15; END_IF;
END_REGION

REGION Network 3 (SCL): Copy HMI Data
   #ioHMI.ControlWord.StepNO := #ioOP[#ioHMI.OP_Select].StepNO[#ioHMI.PageCount];
   #ioHMI.ControlWord.FaultCode := #ioOP[#ioHMI.OP_Select].FaultCode[#ioHMI.PageCount];
   #ioHMI.ControlWord.Busy := #ioOP[#ioHMI.OP_Select].Busy[#ioHMI.PageCount];
   #ioHMI.ControlWord.ResultOK := #ioOP[#ioHMI.OP_Select].ResultOK[#ioHMI.PageCount];
   #ioHMI.ControlWord.ResultNG := #ioOP[#ioHMI.OP_Select].ResultNG[#ioHMI.PageCount];
   IF NOT #iManualMode THEN
       #ioHMI.Enable := 0;
   END_IF;
END_REGION

REGION Network 4: HMI.ControlWord.Trigger / ControlWord.Trigger
   RUNG wire#powerrail
      Contact( #iManualMode )
      Contact( "OneMES_ControlData".HMI.Enable )
      P_Contact(operand := #ioHMI.ControlWord.Trigger, bit := #ioPluse)
      S_Coil( #ioOP[#ioHMI.OP_Select].Trigger[#ioHMI.PageCount] )
   END_RUNG
   // the same network as SCL:
   #_w1 := #iManualMode AND "OneMES_ControlData".HMI.Enable AND #ioHMI.ControlWord.Trigger AND NOT #ioPluse;   // rising edge of #ioHMI.ControlWord.Trigger
   #ioPluse := #ioHMI.ControlWord.Trigger;
   IF #_w1 THEN #ioOP[#ioHMI.OP_Select].Trigger[#ioHMI.PageCount] := TRUE; END_IF;
END_REGION

REGION Network 5: OP Limit / MsgDisplay.OP_Sel Limit
   RUNG wire#powerrail
      Contact( TRUE )
      wire#w1
      { S7_Templates := "SrcType := SInt" } GT_Contact(in1 := "OneMES_ControlData".MsgDisplay.OP_Sel, in2 := #iOP_Sum)
      Move(in := 1, out1 => "OneMES_ControlData".MsgDisplay.OP_Sel)
   END_RUNG
   RUNG wire#w1
      { S7_Templates := "SrcType := SInt" } LT_Contact(in1 := "OneMES_ControlData".HMI.OP_Select, in2 := 1)
      Move(in := #iOP_Sum, out1 => "OneMES_ControlData".MsgDisplay.OP_Sel)
   END_RUNG
   // the same network as SCL:
   IF TRUE AND ("OneMES_ControlData".MsgDisplay.OP_Sel > #iOP_Sum) THEN
       "OneMES_ControlData".MsgDisplay.OP_Sel := 1;
   END_IF;
   IF TRUE AND ("OneMES_ControlData".HMI.OP_Select < 1) THEN
       "OneMES_ControlData".MsgDisplay.OP_Sel := #iOP_Sum;
   END_IF;
END_REGION

REGION Network 6 (SCL)
   CASE "OneMES_ControlData".HMI.OP_Select OF
       1:
           "OneMES_ControlData".MsgDisplay.DB_NO1 := 2001;
           "OneMES_ControlData".MsgDisplay.DB_NO2 := 2002;
           "OneMES_ControlData".MsgDisplay.DB_NO3 := 2003;
           "OneMES_ControlData".MsgDisplay.DB_NO4 := 2004;
           "OneMES_ControlData".MsgDisplay.DB_NO5 := 2005;
           "OneMES_ControlData".MsgDisplay.DB_NO6 := 2006;
           "OneMES_ControlData".MsgDisplay.DB_NO7 := 2007;

       2:
           "OneMES_ControlData".MsgDisplay.DB_NO1 := 2011;
           "OneMES_ControlData".MsgDisplay.DB_NO2 := 2012;
           "OneMES_ControlData".MsgDisplay.DB_NO3 := 2013;
           "OneMES_ControlData".MsgDisplay.DB_NO4 := 2014;
           "OneMES_ControlData".MsgDisplay.DB_NO5 := 2015;
           "OneMES_ControlData".MsgDisplay.DB_NO6 := 2016;
           "OneMES_ControlData".MsgDisplay.DB_NO7 := 2017;

       3:
           "OneMES_ControlData".MsgDisplay.DB_NO1 := 2021;
           "OneMES_ControlData".MsgDisplay.DB_NO2 := 2022;
           "OneMES_ControlData".MsgDisplay.DB_NO3 := 2023;
           "OneMES_ControlData".MsgDisplay.DB_NO4 := 2024;
           "OneMES_ControlData".MsgDisplay.DB_NO5 := 2025;
           "OneMES_ControlData".MsgDisplay.DB_NO6 := 2026;
           "OneMES_ControlData".MsgDisplay.DB_NO7 := 2027;

       4:
           "OneMES_ControlData".MsgDisplay.DB_NO1 := 2031;
           "OneMES_ControlData".MsgDisplay.DB_NO2 := 2032;
           "OneMES_ControlData".MsgDisplay.DB_NO3 := 2033;
           "OneMES_ControlData".MsgDisplay.DB_NO4 := 2034;
           "OneMES_ControlData".MsgDisplay.DB_NO5 := 2035;
           "OneMES_ControlData".MsgDisplay.DB_NO6 := 2036;
           "OneMES_ControlData".MsgDisplay.DB_NO7 := 2037;

       5:
           "OneMES_ControlData".MsgDisplay.DB_NO1 := 2041;
           "OneMES_ControlData".MsgDisplay.DB_NO2 := 2042;
           "OneMES_ControlData".MsgDisplay.DB_NO3 := 2043;
           "OneMES_ControlData".MsgDisplay.DB_NO4 := 2044;
           "OneMES_ControlData".MsgDisplay.DB_NO5 := 2045;
           "OneMES_ControlData".MsgDisplay.DB_NO6 := 2046;
           "OneMES_ControlData".MsgDisplay.DB_NO7 := 2047;

       // ELSE  "OneMES_ControlData".MsgDisplay.OP_Sel :=1
       //     ;
   END_CASE;
END_REGION

REGION Network 7 (SCL): MES Msg Display
   CASE "OneMES_ControlData".HMI.OP_Select OF
       1:
           "OneMES_ControlData".MsgDisplay.PLC_RequestTimeOutCount_Offset := 6; 
          "OneMES_ControlData".MsgDisplay.PLC_RequestTransaction_ID_Offset := 8;
          "OneMES_ControlData".MsgDisplay.PLC_RequestSignal_Offset := 12;
          "OneMES_ControlData".MsgDisplay.MES_ResponseError_ID_Offset := 14;
          "OneMES_ControlData".MsgDisplay.MES_ResponseSignal_Offset := 16;

      2:
          "OneMES_ControlData".MsgDisplay.PLC_RequestTimeOutCount_Offset := 18;
          "OneMES_ControlData".MsgDisplay.PLC_RequestTransaction_ID_Offset := 8;
          "OneMES_ControlData".MsgDisplay.PLC_RequestSignal_Offset := 20;
          "OneMES_ControlData".MsgDisplay.MES_ResponseError_ID_Offset := 22;
          "OneMES_ControlData".MsgDisplay.MES_ResponseSignal_Offset := 24;

      3:
          "OneMES_ControlData".MsgDisplay.PLC_RequestTimeOutCount_Offset := 26;
          "OneMES_ControlData".MsgDisplay.PLC_RequestTransaction_ID_Offset := 28;
          "OneMES_ControlData".MsgDisplay.PLC_RequestSignal_Offset := 32;
          "OneMES_ControlData".MsgDisplay.MES_ResponseError_ID_Offset := 34;
          "OneMES_ControlData".MsgDisplay.MES_ResponseSignal_Offset := 36;

      4:
          "OneMES_ControlData".MsgDisplay.PLC_RequestTimeOutCount_Offset := 38;
          "OneMES_ControlData".MsgDisplay.PLC_RequestTransaction_ID_Offset := 40;
          "OneMES_ControlData".MsgDisplay.PLC_RequestSignal_Offset := 44;
          "OneMES_ControlData".MsgDisplay.MES_ResponseError_ID_Offset := 46;
          "OneMES_ControlData".MsgDisplay.MES_ResponseSignal_Offset := 48;

      5:
          "OneMES_ControlData".MsgDisplay.PLC_RequestTimeOutCount_Offset := 50;
          "OneMES_ControlData".MsgDisplay.PLC_RequestTransaction_ID_Offset := 52;
          "OneMES_ControlData".MsgDisplay.PLC_RequestSignal_Offset := 56;
          "OneMES_ControlData".MsgDisplay.MES_ResponseError_ID_Offset := 58;
          "OneMES_ControlData".MsgDisplay.MES_ResponseSignal_Offset := 60;

      6:
          "OneMES_ControlData".MsgDisplay.PLC_RequestTimeOutCount_Offset := 62;
          "OneMES_ControlData".MsgDisplay.PLC_RequestTransaction_ID_Offset := 64;
          "OneMES_ControlData".MsgDisplay.PLC_RequestSignal_Offset := 68;
          "OneMES_ControlData".MsgDisplay.MES_ResponseError_ID_Offset := 70;
          "OneMES_ControlData".MsgDisplay.MES_ResponseSignal_Offset := 72;

      7:
          "OneMES_ControlData".MsgDisplay.PLC_RequestTimeOutCount_Offset := 74;
          "OneMES_ControlData".MsgDisplay.PLC_RequestTransaction_ID_Offset := 76;
          "OneMES_ControlData".MsgDisplay.PLC_RequestSignal_Offset := 80;
          "OneMES_ControlData".MsgDisplay.MES_ResponseError_ID_Offset := 82;
          "OneMES_ControlData".MsgDisplay.MES_ResponseSignal_Offset := 84;

      8:
          "OneMES_ControlData".MsgDisplay.PLC_RequestTimeOutCount_Offset := 86;
          "OneMES_ControlData".MsgDisplay.PLC_RequestTransaction_ID_Offset := 88;
          "OneMES_ControlData".MsgDisplay.PLC_RequestSignal_Offset := 92;
          "OneMES_ControlData".MsgDisplay.MES_ResponseError_ID_Offset := 94;
          "OneMES_ControlData".MsgDisplay.MES_ResponseSignal_Offset := 96;

      9:
          "OneMES_ControlData".MsgDisplay.PLC_RequestTimeOutCount_Offset := 98;
          "OneMES_ControlData".MsgDisplay.PLC_RequestTransaction_ID_Offset := 100;
          "OneMES_ControlData".MsgDisplay.PLC_RequestSignal_Offset := 104;
          "OneMES_ControlData".MsgDisplay.MES_ResponseError_ID_Offset := 106;
          "OneMES_ControlData".MsgDisplay.MES_ResponseSignal_Offset := 96;

      10:
          "OneMES_ControlData".MsgDisplay.PLC_RequestTimeOutCount_Offset := 108;
          "OneMES_ControlData".MsgDisplay.PLC_RequestTransaction_ID_Offset := 110;
          "OneMES_ControlData".MsgDisplay.PLC_RequestSignal_Offset := 114;
          "OneMES_ControlData".MsgDisplay.MES_ResponseError_ID_Offset := 116;
          "OneMES_ControlData".MsgDisplay.MES_ResponseSignal_Offset := 118;

      11:
          "OneMES_ControlData".MsgDisplay.PLC_RequestTimeOutCount_Offset := 120;
          "OneMES_ControlData".MsgDisplay.PLC_RequestTransaction_ID_Offset := 122;
          "OneMES_ControlData".MsgDisplay.PLC_RequestSignal_Offset := 126;
          "OneMES_ControlData".MsgDisplay.MES_ResponseError_ID_Offset := 128;
          "OneMES_ControlData".MsgDisplay.MES_ResponseSignal_Offset := 130;

      12:
          "OneMES_ControlData".MsgDisplay.PLC_RequestTimeOutCount_Offset := 132;
          "OneMES_ControlData".MsgDisplay.PLC_RequestTransaction_ID_Offset := 134;
          "OneMES_ControlData".MsgDisplay.PLC_RequestSignal_Offset := 138;
          "OneMES_ControlData".MsgDisplay.MES_ResponseError_ID_Offset := 140;
          "OneMES_ControlData".MsgDisplay.MES_ResponseSignal_Offset := 142;

      13:
          "OneMES_ControlData".MsgDisplay.PLC_RequestTimeOutCount_Offset := 152;
          "OneMES_ControlData".MsgDisplay.PLC_RequestTransaction_ID_Offset := 154;
          "OneMES_ControlData".MsgDisplay.PLC_RequestSignal_Offset := 158;
          "OneMES_ControlData".MsgDisplay.MES_ResponseError_ID_Offset := 160;
          "OneMES_ControlData".MsgDisplay.MES_ResponseSignal_Offset := 162;

      14:
          "OneMES_ControlData".MsgDisplay.PLC_RequestTimeOutCount_Offset := 170;
          "OneMES_ControlData".MsgDisplay.PLC_RequestTransaction_ID_Offset := 172;
          "OneMES_ControlData".MsgDisplay.PLC_RequestSignal_Offset := 176;
          "OneMES_ControlData".MsgDisplay.MES_ResponseError_ID_Offset := 178;
          "OneMES_ControlData".MsgDisplay.MES_ResponseSignal_Offset := 180;

      15:
          "OneMES_ControlData".MsgDisplay.PLC_RequestTimeOutCount_Offset := 6;
          "OneMES_ControlData".MsgDisplay.PLC_RequestTransaction_ID_Offset := 8;
          "OneMES_ControlData".MsgDisplay.PLC_RequestSignal_Offset := 12;
          "OneMES_ControlData".MsgDisplay.MES_ResponseError_ID_Offset := 14;
          "OneMES_ControlData".MsgDisplay.MES_ResponseSignal_Offset := 16;

       // ELSE  
       //     "OneMES_ControlData".MsgDisplay.Process_Sel:=1   ;
   END_CASE;
END_REGION
END_FUNCTION

FUNCTION_BLOCK "FB_Pos16"   // FB30141, LAD
{ S7_Optimized_Access := 'TRUE' }
// stored: AutoNumber false, MemoryReserve 100, SetENOAutomatically false
   VAR_INPUT
      Opmode { ExternalAccessible := 'False'; ExternalVisible := 'False'; ExternalWritable := 'False'} : "OPMODE_OUT_UDT";
      TO_PosAxis : TO_PositioningAxis;
      I_iNum_Abspos : Int;
      I_bMan_Enable : Bool;
   END_VAR
   VAR_IN_OUT
      Ds_Pos16 : "sPos16";
   END_VAR
   VAR
      instAxis01 { ExternalAccessible := 'False'; ExternalVisible := 'False'; ExternalWritable := 'False'} : "LAxisCtrl_PosAxis";
      instShearAxisStatus { S7_SetPoint := 'True'} : "LAxisCtrl_GetAxisStatusWord";
      RT_Reset { S7_SetPoint := 'True'} : R_TRIG;
      RT_PB { ExternalAccessible := 'False'; ExternalVisible := 'False'; ExternalWritable := 'False'} : Array[0..19] of R_TRIG;   // Störungen / Alarms
      FT_PB { ExternalAccessible := 'False'; ExternalVisible := 'False'; ExternalWritable := 'False'; S7_SetPoint := 'True'} : Array[0..19] of F_TRIG;   // Störungen unterdrücken, Belegung identisch mit "Alarm" / Hide Alarms, identical with "Alarm"
      TON_PB { ExternalAccessible := 'False'; ExternalVisible := 'False'; ExternalWritable := 'False'} : Array[0..19] of TON_TIME;   // Fallende Flanke / Falling edge
      TOF_PB { ExternalAccessible := 'False'; ExternalVisible := 'False'; ExternalWritable := 'False'} : Array[0..19] of TOF_TIME;   // Negativer Impuls / Negative pulse
      i { S7_SetPoint := 'True'} : Int;
      temp_cmd_bEnableAxis { ExternalAccessible := 'False'; ExternalVisible := 'False'; ExternalWritable := 'False'} : Bool;
      temp_cmd_bresetAxis { ExternalAccessible := 'False'; ExternalVisible := 'False'; ExternalWritable := 'False'} : Bool;
      temp_cmd_bjogForward { ExternalAccessible := 'False'; ExternalVisible := 'False'; ExternalWritable := 'False'} : Bool;
      temp_cmd_bjogBackward { ExternalAccessible := 'False'; ExternalVisible := 'False'; ExternalWritable := 'False'} : Bool;
      temp_cmd_bmoveVelocity { ExternalAccessible := 'False'; ExternalVisible := 'False'; ExternalWritable := 'False'} : Bool;
      temp_cmd_bstop { ExternalAccessible := 'False'; ExternalVisible := 'False'; ExternalWritable := 'False'} : Bool;
      temp_cmd_bfastStop { ExternalAccessible := 'False'; ExternalVisible := 'False'; ExternalWritable := 'False'} : Bool;
      temp_cmd_bhoming { ExternalAccessible := 'False'; ExternalVisible := 'False'; ExternalWritable := 'False'} : Bool;
      temp_cmd_bGoToPos { ExternalAccessible := 'False'; ExternalVisible := 'False'; ExternalWritable := 'False'} : Array[0..16] of Bool;
      temp_cmd_iGoToPos : Word;
      temp_cmd_bCallAbsPos : Bool;
      temp_cmd_bRelPos : Bool;
      temp_Para_rJog_Speed { ExternalAccessible := 'False'; ExternalVisible := 'False'; ExternalWritable := 'False'} : LReal;
      temp_configuration { ExternalAccessible := 'False'; ExternalVisible := 'False'; ExternalWritable := 'False'} : "LAxisCtrl_typeAxisConfig";   // Diagnostics structure
      temp_Status { ExternalAccessible := 'False'; ExternalVisible := 'False'; ExternalWritable := 'False'} : Word;
      temp_AxisEnabled { ExternalAccessible := 'False'; ExternalVisible := 'False'; ExternalWritable := 'False'} : Bool;
      temp_CommandBusy { ExternalAccessible := 'False'; ExternalVisible := 'False'; ExternalWritable := 'False'} : Bool;
      temp_CommandDone { ExternalAccessible := 'False'; ExternalVisible := 'False'; ExternalWritable := 'False'} : Bool;
      temp_CommandAborted { ExternalAccessible := 'False'; ExternalVisible := 'False'; ExternalWritable := 'False'} : Bool;
      temp_InVelocity { ExternalAccessible := 'False'; ExternalVisible := 'False'; ExternalWritable := 'False'} : Bool;
      temp_jogSelected { ExternalAccessible := 'False'; ExternalVisible := 'False'; ExternalWritable := 'False'} : Bool;
      tempPosAbsoluteSelected { ExternalAccessible := 'False'; ExternalVisible := 'False'; ExternalWritable := 'False'} : Bool;
      temp_diagnostics { ExternalAccessible := 'False'; ExternalVisible := 'False'; ExternalWritable := 'False'} : "LAxisCtrl_typeDiagnostics";
      temp_stop_Dec { ExternalAccessible := 'False'; ExternalVisible := 'False'; ExternalWritable := 'False'} : LReal;
      temp_faststop_Dec { ExternalAccessible := 'False'; ExternalVisible := 'False'; ExternalWritable := 'False'} : LReal;
      temp_cmd_bGoToPosAll : Bool;
      temp_iFBStatus : Word;
      temp_iMCStatus : Word;
      old_iFBStatus : Word;
      old_iMCStatus : Word;
   END_VAR
BEGIN

REGION Network 1
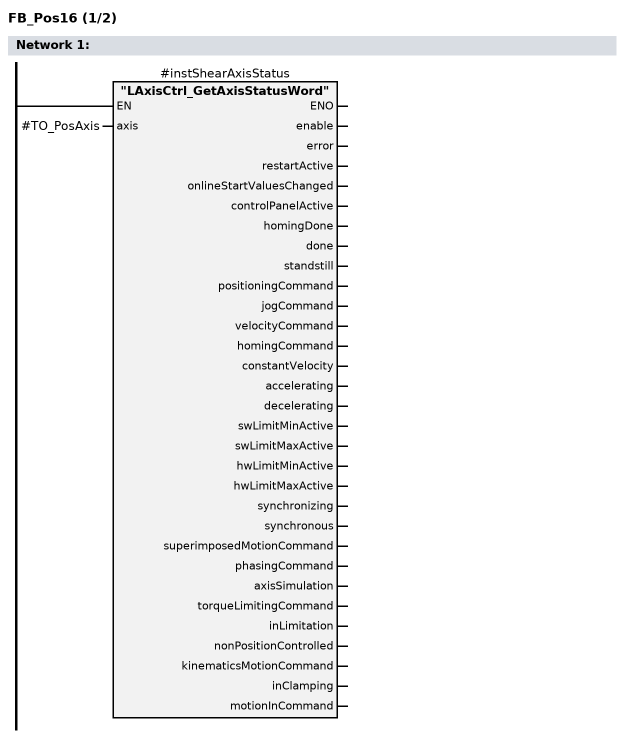
   RUNG wire#powerrail
      #instShearAxisStatus(axis := #TO_PosAxis, enable =>, error =>, restartActive =>, onlineStartValuesChanged =>, controlPanelActive =>, homingDone =>, done =>, standstill =>, positioningCommand =>, jogCommand =>, velocityCommand =>, homingCommand =>, constantVelocity =>, accelerating =>, decelerating =>, swLimitMinActive =>, swLimitMaxActive =>, hwLimitMinActive =>, hwLimitMaxActive =>, synchronizing =>, synchronous =>, superimposedMotionCommand =>, phasingCommand =>, axisSimulation =>, torqueLimitingCommand =>, inLimitation =>, nonPositionControlled =>, kinematicsMotionCommand =>, inClamping =>, motionInCommand =>)
   END_RUNG
   // the same network as SCL:
   #instShearAxisStatus(axis := #TO_PosAxis);   // "LAxisCtrl_GetAxisStatusWord"
END_REGION

REGION Network 2: LAxisCtrl
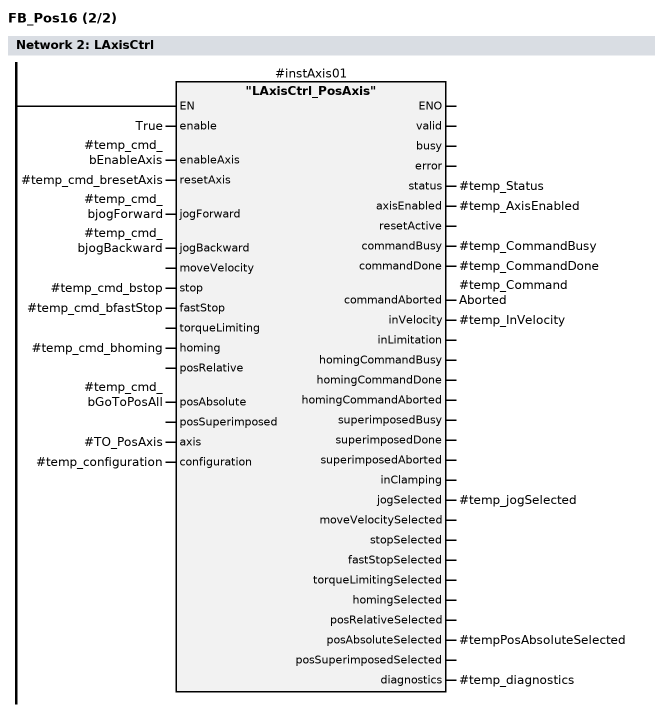
   RUNG wire#powerrail
      #instAxis01(enable := True, enableAxis := #temp_cmd_bEnableAxis, resetAxis := #temp_cmd_bresetAxis, jogForward := #temp_cmd_bjogForward, jogBackward := #temp_cmd_bjogBackward, moveVelocity :=, stop := #temp_cmd_bstop, fastStop := #temp_cmd_bfastStop, torqueLimiting :=, homing := #temp_cmd_bhoming, posRelative :=, posAbsolute := #temp_cmd_bGoToPosAll, posSuperimposed :=, axis := #TO_PosAxis, configuration := #temp_configuration, valid =>, busy =>, error =>, status => #temp_Status, axisEnabled => #temp_AxisEnabled, resetActive =>, commandBusy => #temp_CommandBusy, commandDone => #temp_CommandDone, commandAborted => #temp_CommandAborted, inVelocity => #temp_InVelocity, inLimitation =>, homingCommandBusy =>, homingCommandDone =>, homingCommandAborted =>, superimposedBusy =>, superimposedDone =>, superimposedAborted =>, inClamping =>, jogSelected => #temp_jogSelected, moveVelocitySelected =>, stopSelected =>, fastStopSelected =>, torqueLimitingSelected =>, homingSelected =>, posRelativeSelected =>, posAbsoluteSelected => #tempPosAbsoluteSelected, posSuperimposedSelected =>, diagnostics => #temp_diagnostics)
   END_RUNG
   // the same network as SCL:
   #instAxis01(enable := True,   // "LAxisCtrl_PosAxis"
               enableAxis := #temp_cmd_bEnableAxis,
               resetAxis := #temp_cmd_bresetAxis,
               jogForward := #temp_cmd_bjogForward,
               jogBackward := #temp_cmd_bjogBackward,
               stop := #temp_cmd_bstop,
               fastStop := #temp_cmd_bfastStop,
               homing := #temp_cmd_bhoming,
               posAbsolute := #temp_cmd_bGoToPosAll,
               axis := #TO_PosAxis,
               configuration := #temp_configuration,
               status => #temp_Status,
               axisEnabled => #temp_AxisEnabled,
               commandBusy => #temp_CommandBusy,
               commandDone => #temp_CommandDone,
               commandAborted => #temp_CommandAborted,
               inVelocity => #temp_InVelocity,
               jogSelected => #temp_jogSelected,
               posAbsoluteSelected => #tempPosAbsoluteSelected,
               diagnostics => #temp_diagnostics);
END_REGION

REGION Network 3 (SCL): input
   #temp_cmd_bEnableAxis  := #Ds_Pos16.I_CMD_bEnableAxis OR (#Ds_Pos16.I_HMI_bEnableAxis AND #I_bMan_Enable);
   #temp_cmd_bresetAxis   := #Ds_Pos16.I_CMD_bResetAxis;
   #temp_cmd_bjogForward  := #Ds_Pos16.I_InLock_bjogForward AND (#Ds_Pos16.I_CMD_bjogForward OR (#Ds_Pos16.I_HMI_bjogForward AND #I_bMan_Enable));
   #temp_cmd_bjogBackward := #Ds_Pos16.I_InLock_bjogBackward AND (#Ds_Pos16.I_CMD_bjogBackward OR (#Ds_Pos16.I_HMI_bjogBackward AND #I_bMan_Enable));
   #temp_cmd_bstop        := #Ds_Pos16.I_CMD_bstop OR (#Ds_Pos16.I_HMI_bstop AND #I_bMan_Enable);
   #temp_cmd_bfastStop    := #Ds_Pos16.I_CMD_bfastStop;
   #temp_cmd_bhoming      := #Ds_Pos16.I_InLock_bHoming AND (#Ds_Pos16.I_CMD_bHoming OR #Ds_Pos16.I_HMI_bHoming);
END_REGION

REGION Network 4 (SCL): Configuration
   #Ds_Pos16.I_Para_rJog_Speed[0] := 10.0;
   #Ds_Pos16.I_Para_rMV_Speed[0]  := 10.0;
   #Ds_Pos16.I_Para_rStop_Dec[0]  := 20.0;
   #Ds_Pos16.I_Para_rEStop_Dec[0] := 50.0;

   #Ds_Pos16.I_Para_rJog_Speed[1] := 10.0 * #Ds_Pos16.I_Para_rJog_Speed[0];
   #Ds_Pos16.I_Para_rJog_Speed[2] := 10.0 * #Ds_Pos16.I_Para_rJog_Speed[0];
   #Ds_Pos16.I_Para_rMV_Speed[1] := 10.0 * #Ds_Pos16.I_Para_rMV_Speed[0];
   #Ds_Pos16.I_Para_rMV_Speed[2] := 10.0 * #Ds_Pos16.I_Para_rMV_Speed[0];
   #Ds_Pos16.I_Para_rStop_Dec[1] := 100.0 * #Ds_Pos16.I_Para_rStop_Dec[0];
   #Ds_Pos16.I_Para_rEStop_Dec[1] := 100.0 * #Ds_Pos16.I_Para_rEStop_Dec[0];

   IF #temp_configuration.jog.velocity <> #Ds_Pos16.I_Para_rJog_Speed[0] OR
       #temp_configuration.jog.acceleration <> #Ds_Pos16.I_Para_rJog_Speed[1] OR
       #temp_configuration.jog.deceleration <> #Ds_Pos16.I_Para_rJog_Speed[2] OR
       #temp_configuration.moveVelocity.acceleration <> #Ds_Pos16.I_Para_rMV_Speed[0] OR
       #temp_configuration.moveVelocity.deceleration <> #Ds_Pos16.I_Para_rMV_Speed[1] OR
       #temp_configuration.moveVelocity.acceleration <> #Ds_Pos16.I_Para_rMV_Speed[2] OR
       #temp_configuration.stop.deceleration <> #Ds_Pos16.I_Para_rStop_Dec[0] OR
       #temp_configuration.stop.jerk <> #Ds_Pos16.I_Para_rStop_Dec[1] OR
       #temp_configuration.fastStop.deceleration <> #Ds_Pos16.I_Para_rEStop_Dec[0] OR
       #temp_configuration.fastStop.jerk <> #Ds_Pos16.I_Para_rEStop_Dec[1]
   THEN
       // Jog
       #temp_configuration.jog.velocity := #Ds_Pos16.I_Para_rJog_Speed[0];
       #temp_configuration.jog.acceleration := #Ds_Pos16.I_Para_rJog_Speed[1];
       #temp_configuration.jog.deceleration := #Ds_Pos16.I_Para_rJog_Speed[2];
       // Move
       #temp_configuration.moveVelocity.velocity := #Ds_Pos16.I_Para_rMV_Speed[0];
       #temp_configuration.moveVelocity.acceleration := #Ds_Pos16.I_Para_rMV_Speed[1];
       #temp_configuration.moveVelocity.deceleration := #Ds_Pos16.I_Para_rMV_Speed[2];
       // Stop   
       #temp_configuration.stop.deceleration := #Ds_Pos16.I_Para_rStop_Dec[0];
       #temp_configuration.stop.jerk := #Ds_Pos16.I_Para_rStop_Dec[1];
       //faststoo
       #temp_configuration.fastStop.deceleration := #Ds_Pos16.I_Para_rEStop_Dec[0];
       #temp_configuration.fastStop.jerk := #Ds_Pos16.I_Para_rEStop_Dec[1];
   END_IF;

   // Homing
   #temp_configuration.homing.mode := 0;//I_iHomeMode
   #temp_configuration.homing.position := 0;//I_iHomePos

   //abspos
   FOR #i := 1 TO 16 DO
       #Ds_Pos16.I_Para_rAcc_Set[#i] := 10.0 * #Ds_Pos16.I_Para_rSpeed_Abs[0];
       #Ds_Pos16.I_Para_rDec_Set[#i] := 10.0 * #Ds_Pos16.I_Para_rSpeed_Abs[0];
       #Ds_Pos16.I_Para_rJerk_Set[#i] := 100.0 * #Ds_Pos16.I_Para_rSpeed_Abs[0];
   END_FOR;


   //#temp_posAbsolute := (#Ds_Pos16.I_CMD_iGoToPos <> 16#0);
   #temp_cmd_bGoToPos[1] := ((#Opmode.Automatic_active=1 AND #Ds_Pos16.I_CMD_iGoToPos = 1) OR (#Opmode.Manual_active AND #Ds_Pos16.I_HMI_iGoToPos = 1)) AND #Ds_Pos16.I_InLock_bGoToPos[1];
   #temp_cmd_bGoToPos[2] := ((#Opmode.Automatic_active=1 AND #Ds_Pos16.I_CMD_iGoToPos = 2) OR (#Opmode.Manual_active AND  #Ds_Pos16.I_HMI_iGoToPos = 2)) AND #Ds_Pos16.I_InLock_bGoToPos[2];
   #temp_cmd_bGoToPos[3] := ((#Opmode.Automatic_active=1 AND #Ds_Pos16.I_CMD_iGoToPos = 3) OR (#Opmode.Manual_active AND  #Ds_Pos16.I_HMI_iGoToPos = 3)) AND #Ds_Pos16.I_InLock_bGoToPos[3];
   #temp_cmd_bGoToPos[4] := ((#Opmode.Automatic_active=1 AND #Ds_Pos16.I_CMD_iGoToPos = 4) OR (#Opmode.Manual_active AND  #Ds_Pos16.I_HMI_iGoToPos = 4)) AND #Ds_Pos16.I_InLock_bGoToPos[4];
   #temp_cmd_bGoToPos[5] := ((#Opmode.Automatic_active=1 AND #Ds_Pos16.I_CMD_iGoToPos = 5) OR (#Opmode.Manual_active AND  #Ds_Pos16.I_HMI_iGoToPos = 5)) AND #Ds_Pos16.I_InLock_bGoToPos[5];
   #temp_cmd_bGoToPos[6] := ((#Opmode.Automatic_active=1 AND #Ds_Pos16.I_CMD_iGoToPos = 6) OR (#Opmode.Manual_active AND  #Ds_Pos16.I_HMI_iGoToPos = 6)) AND #Ds_Pos16.I_InLock_bGoToPos[6];
   #temp_cmd_bGoToPos[7] := ((#Opmode.Automatic_active=1 AND #Ds_Pos16.I_CMD_iGoToPos = 7) OR (#Opmode.Manual_active AND  #Ds_Pos16.I_HMI_iGoToPos = 7)) AND #Ds_Pos16.I_InLock_bGoToPos[7];
   #temp_cmd_bGoToPos[8] := ((#Opmode.Automatic_active=1 AND #Ds_Pos16.I_CMD_iGoToPos = 8) OR (#Opmode.Manual_active AND  #Ds_Pos16.I_HMI_iGoToPos = 8)) AND #Ds_Pos16.I_InLock_bGoToPos[8];
   #temp_cmd_bGoToPos[9] := ((#Opmode.Automatic_active=1 AND #Ds_Pos16.I_CMD_iGoToPos = 9) OR (#Opmode.Manual_active AND  #Ds_Pos16.I_HMI_iGoToPos = 9)) AND #Ds_Pos16.I_InLock_bGoToPos[9];
   #temp_cmd_bGoToPos[10] := ((#Opmode.Automatic_active=1 AND #Ds_Pos16.I_CMD_iGoToPos = 10) OR (#Opmode.Manual_active AND  #Ds_Pos16.I_HMI_iGoToPos = 10)) AND #Ds_Pos16.I_InLock_bGoToPos[10];
   #temp_cmd_bGoToPos[11] := ((#Opmode.Automatic_active=1 AND #Ds_Pos16.I_CMD_iGoToPos = 11) OR (#Opmode.Manual_active AND  #Ds_Pos16.I_HMI_iGoToPos = 11)) AND #Ds_Pos16.I_InLock_bGoToPos[11];
   #temp_cmd_bGoToPos[12] := ((#Opmode.Automatic_active=1 AND #Ds_Pos16.I_CMD_iGoToPos = 12) OR (#Opmode.Manual_active AND  #Ds_Pos16.I_HMI_iGoToPos = 12)) AND #Ds_Pos16.I_InLock_bGoToPos[12];
   #temp_cmd_bGoToPos[13] := ((#Opmode.Automatic_active=1 AND #Ds_Pos16.I_CMD_iGoToPos = 13) OR (#Opmode.Manual_active AND  #Ds_Pos16.I_HMI_iGoToPos = 13)) AND #Ds_Pos16.I_InLock_bGoToPos[13];
   #temp_cmd_bGoToPos[14] := ((#Opmode.Automatic_active=1 AND #Ds_Pos16.I_CMD_iGoToPos = 14) OR (#Opmode.Manual_active AND  #Ds_Pos16.I_HMI_iGoToPos = 14)) AND #Ds_Pos16.I_InLock_bGoToPos[14];
   #temp_cmd_bGoToPos[15] := ((#Opmode.Automatic_active=1 AND #Ds_Pos16.I_CMD_iGoToPos = 15) OR (#Opmode.Manual_active AND  #Ds_Pos16.I_HMI_iGoToPos = 15)) AND #Ds_Pos16.I_InLock_bGoToPos[15];
   #temp_cmd_bGoToPos[16] := ((#Opmode.Automatic_active=1 AND #Ds_Pos16.I_CMD_iGoToPos = 16) OR (#Opmode.Manual_active AND  #Ds_Pos16.I_HMI_iGoToPos = 16)) AND #Ds_Pos16.I_InLock_bGoToPos[16];

   #temp_cmd_bGoToPosAll := #temp_cmd_bGoToPos[1] OR #temp_cmd_bGoToPos[2] OR #temp_cmd_bGoToPos[3] OR #temp_cmd_bGoToPos[4]
   OR #temp_cmd_bGoToPos[5] OR #temp_cmd_bGoToPos[6] OR #temp_cmd_bGoToPos[7] OR #temp_cmd_bGoToPos[8]
   OR #temp_cmd_bGoToPos[9] OR #temp_cmd_bGoToPos[10] OR #temp_cmd_bGoToPos[11] OR #temp_cmd_bGoToPos[12]
   OR #temp_cmd_bGoToPos[13] OR #temp_cmd_bGoToPos[14] OR #temp_cmd_bGoToPos[15] OR #temp_cmd_bGoToPos[16]
   ;
   //#temp_posAbsolute :=
   //#Ds_Pos16.I_bGoToPos[0] OR #Ds_Pos16.I_bGoToPos[1] OR #Ds_Pos16.I_bGoToPos[2] OR #Ds_Pos16.I_bGoToPos[3] OR
   //#Ds_Pos16.I_bGoToPos[4] OR #Ds_Pos16.I_bGoToPos[5] OR #Ds_Pos16.I_bGoToPos[6] OR #Ds_Pos16.I_bGoToPos[7] OR
   //#Ds_Pos16.I_bGoToPos[8] OR #Ds_Pos16.I_bGoToPos[9] OR #Ds_Pos16.I_bGoToPos[10] OR #Ds_Pos16.I_bGoToPos[11] OR
   //#Ds_Pos16.I_bGoToPos[12] OR #Ds_Pos16.I_bGoToPos[13] OR #Ds_Pos16.I_bGoToPos[14] OR #Ds_Pos16.I_bGoToPos[15];

   FOR #i := 1 TO 16 DO
   //    #RT_PB[#i](CLK := #Ds_Pos16.I_bGoToPos[#i]);
       #RT_PB[#i](CLK := #temp_cmd_bGoToPos[#i]);

       IF #RT_PB[#i].Q THEN
           #temp_configuration.posAbsolute.position := #Ds_Pos16.I_Para_rPos_Abs[#i];
           #temp_configuration.posAbsolute.velocity := #Ds_Pos16.I_Para_rSpeed_Abs[#i];
           #temp_configuration.posAbsolute.direction := 3;//temp_posAbsolute_direction

           #temp_configuration.posAbsolute.acceleration := #Ds_Pos16.I_Para_rAcc_Set[#i];
           #temp_configuration.posAbsolute.deceleration := #Ds_Pos16.I_Para_rDec_Set[#i];
           #temp_configuration.posAbsolute.jerk := #Ds_Pos16.I_Para_rJerk_Set[#i];

       END_IF;
   END_FOR;
END_REGION

REGION Network 5 (SCL): output
   #Ds_Pos16.O_Status_bAxisReady := true;//#TO_PosAxis.StatusWord.%X1;
   #Ds_Pos16.O_Status_bAxisEnabled := #temp_AxisEnabled;
   #Ds_Pos16.O_Status_bjogForward := #temp_cmd_bjogForward;// AND #temp_jogSelected;
   #Ds_Pos16.O_Status_bjogBackward := #temp_cmd_bjogBackward;// AND #temp_jogSelected;
   #Ds_Pos16.O_Status_bHomed := #TO_PosAxis.StatusWord.%X5;
   #Ds_Pos16.O_Status_bAxisError := #TO_PosAxis.StatusWord.%X1;
   #Ds_Pos16.O_Status_rActPos := #TO_PosAxis.ActualPosition;
   #Ds_Pos16.O_Status_rActSpeed := #TO_PosAxis.ActualVelocity;
   #Ds_Pos16.O_Status_iAxisFaultNum := #TO_PosAxis.ErrorDetail.Number;
   //#Ds_Pos16.O_DriveFaultNum
   //#Ds_Pos16.O_Status_iFBStatus := #temp_diagnostics.status;
   //#Ds_Pos16.O_Status_iMCStatus := #temp_diagnostics.subfunctionStatus;
   //#Ds_Pos16.O_Torque
   //#Ds_Pos16.oAxisName  := 

   FOR #i := 0 TO 15 DO
       #Ds_Pos16.O_Status_bAtPos[#i] := "FC_bNearIn"(rAct := #Ds_Pos16.O_Status_rActPos, rTgt := #Ds_Pos16.I_Para_rPos_Abs[#i], rDelta := 1.0, bModule := 0, rModulo := 0);
   END_FOR;

   //#Ds_Pos16.O_bPosDone
   //#Ds_Pos16.O_bPosing
   //#tempPosAbsoluteSelected
END_REGION

REGION Network 6 (SCL): Reset
   #RT_Reset(CLK := #temp_cmd_bresetAxis);
   IF #RT_Reset.Q THEN
       #Ds_Pos16.O_Status_iFBStatus := 16#00;
       #Ds_Pos16.O_Status_iMCStatus := 16#00;
   END_IF;

   #temp_iFBStatus := #temp_diagnostics.status;
   IF #temp_iFBStatus <> #old_iFBStatus THEN
       #Ds_Pos16.O_Status_iFBStatus := #temp_diagnostics.status;
       #old_iFBStatus := #temp_iFBStatus;
   END_IF;
   #temp_iMCStatus := #temp_diagnostics.subfunctionStatus;
   IF #temp_iMCStatus <> #old_iMCStatus THEN
       #Ds_Pos16.O_Status_iFBStatus := #temp_diagnostics.subfunctionStatus;
       #old_iMCStatus := #temp_iMCStatus;
   END_IF;
END_REGION

REGION Network 7 (SCL)
   (*
   FOR #i := 9 TO 16 DO
       IF #I_iNum_Abspos < #i THEN
           #Ds_Pos16.I_InLock_bGoToPos[#i] := false;
       END_IF;
   END_FOR;
   *)
END_REGION
END_FUNCTION_BLOCK

FUNCTION_BLOCK "FB_IO_Map_Disp"
{ S7_Optimized_Access := 'TRUE' }
VERSION : 0.1
   VAR 
      Start_Address_IByte : UInt;
      Start_Address_OByte : UInt;
      Start_Address_SIByte : UDInt := 30000;
      Start_Address_SOByte : UDInt := 30000;
      Loop_I : Int;
      Input : Array[0..15] of Bool;
      SInput : Array[0..15] of Bool;
      Loop_O : Int;
      Output : Array[0..15] of Bool;
      SOutput : Array[0..15] of Bool;
   END_VAR


BEGIN
	
	IF #Start_Address_IByte < 1000 AND #Start_Address_OByte < 1000 THEN
	    FOR #Loop_I := 0 TO 7 DO
	        #Input[#Loop_I] := PEEK_BOOL(area := 16#81, dbNumber := 0, byteOffset := #Start_Address_IByte, bitOffset := #Loop_I);
	        #Input[#Loop_I + 8] := PEEK_BOOL(area := 16#81, dbNumber := 0, byteOffset := #Start_Address_IByte + 1, bitOffset := #Loop_I);
	    END_FOR;
	    FOR #Loop_O := 0 TO 7 DO
	        #Output[#Loop_O] := PEEK_BOOL(area := 16#82, dbNumber := 0, byteOffset := #Start_Address_OByte, bitOffset := #Loop_O);
	        #Output[#Loop_O + 8] := PEEK_BOOL(area := 16#82, dbNumber := 0, byteOffset := #Start_Address_OByte + 1, bitOffset := #Loop_O);
	    END_FOR;
	END_IF;
	
	
	IF #Start_Address_SIByte >= 30000  AND #Start_Address_SOByte >= 30000 THEN
	    FOR #Loop_I := 0 TO 7 DO
	        #SInput[#Loop_I] := PEEK_BOOL(area := 16#81, dbNumber := 0, byteOffset := #Start_Address_SIByte, bitOffset := #Loop_I);
	        #SInput[#Loop_I + 8] := PEEK_BOOL(area := 16#81, dbNumber := 0, byteOffset := #Start_Address_SIByte + 1, bitOffset := #Loop_I);
	    END_FOR;
	    FOR #Loop_O := 0 TO 7 DO
	        #SOutput[#Loop_O] := PEEK_BOOL(area := 16#82, dbNumber := 0, byteOffset := #Start_Address_SOByte, bitOffset := #Loop_O);
	        #SOutput[#Loop_O + 8] := PEEK_BOOL(area := 16#82, dbNumber := 0, byteOffset := #Start_Address_SOByte + 1, bitOffset := #Loop_O);
	    END_FOR;
	END_IF;
	
END_FUNCTION_BLOCK

FUNCTION "LGF_BitsToWord" : Word
{ S7_Optimized_Access := 'TRUE' }
VERSION : 0.1
   VAR_INPUT 
      bit0 : Bool;
      bit1 : Bool;
      bit2 : Bool;
      bit3 : Bool;
      bit4 : Bool;
      bit5 : Bool;
      bit6 : Bool;
      bit7 : Bool;
      bit8 : Bool;
      bit9 : Bool;
      bit10 : Bool;
      bit11 : Bool;
      bit12 : Bool;
      bit13 : Bool;
      bit14 : Bool;
      bit15 : Bool;
   END_VAR


BEGIN
	#LGF_BitsToWord.%X0 := #bit0;
	#LGF_BitsToWord.%X1 := #bit1;
	#LGF_BitsToWord.%X2 := #bit2;
	#LGF_BitsToWord.%X3 := #bit3;
	#LGF_BitsToWord.%X4 := #bit4;
	#LGF_BitsToWord.%X5 := #bit5;
	#LGF_BitsToWord.%X6 := #bit6;
	#LGF_BitsToWord.%X7 := #bit7;
	#LGF_BitsToWord.%X8 := #bit8;
	#LGF_BitsToWord.%X9 := #bit9;
	#LGF_BitsToWord.%X10 := #bit10;
	#LGF_BitsToWord.%X11 := #bit11;
	#LGF_BitsToWord.%X12 := #bit12;
	#LGF_BitsToWord.%X13 := #bit13;
	#LGF_BitsToWord.%X14 := #bit14;
	#LGF_BitsToWord.%X15 := #bit15;
END_FUNCTION

FUNCTION "FC_bNearIn" : Bool
{ S7_Optimized_Access := 'TRUE' }
VERSION : 0.1
   VAR_INPUT 
      rAct : LReal;
      rTgt : LReal;
      rDelta : LReal;
      bModule : Bool;
      rModulo : LReal;
   END_VAR

   VAR_TEMP 
      temppos : LReal;
   END_VAR


BEGIN
	        IF #bModule THEN
	            #temppos := #rTgt - #rAct;
	            
	            WHILE #temppos < -1 * #rModulo / 2 OR #temppos >= #rModulo / 2 DO
	                IF #temppos < -1 * #rModulo / 2 THEN
	                    #temppos := #temppos + #rModulo;
	                END_IF;
	                
	                IF #temppos >= #rModulo / 2 THEN
	                    #temppos := #temppos - #rModulo;
	                END_IF;
	            END_WHILE;
	            
	            #FC_bNearIn := ABS(#temppos) < #rDelta;
	        ELSE
	            
	            #FC_bNearIn := (#rAct >= #rTgt - #rDelta) AND (#rAct <= #rTgt + #rDelta);
	        END_IF;
	        
	        
END_FUNCTION

FUNCTION "FC_AxisChange" : Void
{ S7_Optimized_Access := 'TRUE' }
VERSION : 0.1
   VAR_TEMP 
      i : Int;
   END_VAR


BEGIN
	//切换轴
	(*
	IF "dGlobal".Old_Axis_Select <> "dGlobal".gbo_Axis_Select THEN//刚切换
	    "dStruct_Axis".gs_Axis[#i].I_HMI := "dStruct_Axis".gs_Axis_HMI_Init;
	    
	    "dGlobal".Old_Axis_Select := "dGlobal".gbo_Axis_Select;
	ELSE
	    "dStruct_Axis".gs_Axis["dGlobal".gbo_Axis_Select].I_HMI := "dStruct_Axis".gs_Axis[0].I_HMI;
	 //   "dStruct_Axis".gs_Axis["dGlobal".gbo_Axis_Select].I_CMD := "dStruct_Axis".gs_Axis[0].I_CMD;
	    "dStruct_Axis".gs_Axis["dGlobal".gbo_Axis_Select].I_Para.rJerk_Set[0] := "dStruct_Axis".gs_Axis[0].I_Para.rJerk_Set[0];
	    
	    "dStruct_Axis".gs_Axis[0].I_InLock := "dStruct_Axis".gs_Axis["dGlobal".gbo_Axis_Select].I_InLock;
	    "dStruct_Axis".gs_Axis[0].I_SS := "dStruct_Axis".gs_Axis["dGlobal".gbo_Axis_Select].I_SS;
	    "dStruct_Axis".gs_Axis[0].O_Status := "dStruct_Axis".gs_Axis["dGlobal".gbo_Axis_Select].O_Status;
	
	END_IF;
	*)
	
	//保存显示值到设定 读取设定到显示
	//切换定位段
	IF "dGlobal".Old_Pos_Select <> "dGlobal".gbo_Pos_Select THEN//刚切换
	    "dStruct_Axis".gs_Axis[0].I_Para.rPos_Abs[0]   := "dStruct_Axis".gs_Axis["dGlobal".gbo_Axis_Select].I_Para.rPos_Abs["dGlobal".gbo_Pos_Select];
	    "dStruct_Axis".gs_Axis[0].I_Para.rSpeed_Abs[0] := "dStruct_Axis".gs_Axis["dGlobal".gbo_Axis_Select].I_Para.rSpeed_Abs["dGlobal".gbo_Pos_Select];
	    
	    "dGlobal".Old_Pos_Select := "dGlobal".gbo_Pos_Select;
	ELSE
	    "dStruct_Axis".gs_Axis["dGlobal".gbo_Axis_Select].I_Para.rPos_Abs["dGlobal".gbo_Pos_Select] := "dStruct_Axis".gs_Axis[0].I_Para.rPos_Abs[0];
	    "dStruct_Axis".gs_Axis["dGlobal".gbo_Axis_Select].I_Para.rSpeed_Abs["dGlobal".gbo_Pos_Select] := "dStruct_Axis".gs_Axis[0].I_Para.rSpeed_Abs[0];
	END_IF;
	
	
	
	
	
	
	    
	    
	    
END_FUNCTION

FUNCTION_BLOCK "LAxisCtrl_GetAxisErrorWord"
{ S7_Optimized_Access := 'TRUE' }
AUTHOR : 'tech.team.motioncontrol@siemens.com'
FAMILY : AxisCtrl
VERSION : 1.0
   VAR_INPUT 
      axis {InstructionName := 'TO_SpeedAxis'; LibVersion := '6.0'} : TO_SpeedAxis;
   END_VAR

   VAR_OUTPUT 
      systemFault { ExternalWritable := 'False'; S7_HiddenAssignment := 'HideIfNoParamAssigned'} : Bool;
      configFault { ExternalWritable := 'False'; S7_HiddenAssignment := 'HideIfNoParamAssigned'} : Bool;
      userFault { ExternalWritable := 'False'; S7_HiddenAssignment := 'HideIfNoParamAssigned'} : Bool;
      commandNotAccepted { ExternalWritable := 'False'; S7_HiddenAssignment := 'HideIfNoParamAssigned'} : Bool;
      driveFault { ExternalWritable := 'False'; S7_HiddenAssignment := 'HideIfNoParamAssigned'} : Bool;
      sensorFault { ExternalWritable := 'False'; S7_HiddenAssignment := 'HideIfNoParamAssigned'} : Bool;
      dynamicError { ExternalWritable := 'False'; S7_HiddenAssignment := 'HideIfNoParamAssigned'} : Bool;
      communicationFault { ExternalWritable := 'False'; S7_HiddenAssignment := 'HideIfNoParamAssigned'} : Bool;
      swLimit { ExternalWritable := 'False'; S7_HiddenAssignment := 'HideIfNoParamAssigned'} : Bool;
      hwLimit { ExternalWritable := 'False'; S7_HiddenAssignment := 'HideIfNoParamAssigned'} : Bool;
      homingError { ExternalWritable := 'False'; S7_HiddenAssignment := 'HideIfNoParamAssigned'} : Bool;
      followingErrorFault { ExternalWritable := 'False'; S7_HiddenAssignment := 'HideIfNoParamAssigned'} : Bool;
      positioningFault { ExternalWritable := 'False'; S7_HiddenAssignment := 'HideIfNoParamAssigned'} : Bool;
      peripheralError { ExternalWritable := 'False'; S7_HiddenAssignment := 'HideIfNoParamAssigned'} : Bool;
      synchronousError { ExternalWritable := 'False'; S7_HiddenAssignment := 'HideIfNoParamAssigned'} : Bool;
      adaptionError { ExternalWritable := 'False'; S7_HiddenAssignment := 'HideIfNoParamAssigned'} : Bool;
   END_VAR

   VAR_TEMP 
      tempErrorWord : DWord;
   END_VAR


BEGIN
	//==========================================================================================
	// SIEMENS AG
	// (c)Copyright 2017 All Rights Reserved
	//------------------------------------------------------------------------------------------
	// Library: LAxisCtrl
	// Tested with: S7-1515T-2 PN
	// Engineering: TIA Portal V15
	// Restrictions: ---
	// Requirements: S7-1500/S7-1500T FW 2.5
	// Functionality: The FB is splitting the error word of an axis into bits.
	// Support: tech.team.motioncontrol@siemens.com
	// Note: Parameter comments are only available in language 'English (United States)'
	//------------------------------------------------------------------------------------------
	// Change log table:
	// Version    Date          Expert in charge    Changes applied
	// 01.00.01   04.10.2016    AL                  First released version
	// 01.00.02   29.03.2017    AL                  Added support information
	//===========================================================================================
	
	//----------------------------------------------------------------------------------------------
	// Read errorword
	//----------------------------------------------------------------------------------------------
	#tempErrorWord := #axis.ErrorWord;
	
	//----------------------------------------------------------------------------------------------
	// Write outputs
	//----------------------------------------------------------------------------------------------
	#systemFault := #tempErrorWord.%X0;
	#configFault := #tempErrorWord.%X1;
	#userFault := #tempErrorWord.%X2;
	#commandNotAccepted := #tempErrorWord.%X3;
	#driveFault := #tempErrorWord.%X4;
	#sensorFault := #tempErrorWord.%X5;
	#dynamicError := #tempErrorWord.%X6;
	#communicationFault := #tempErrorWord.%X7;
	#swLimit := #tempErrorWord.%X8;
	#hwLimit := #tempErrorWord.%X9;
	#homingError := #tempErrorWord.%X10;
	#followingErrorFault := #tempErrorWord.%X11;
	#positioningFault := #tempErrorWord.%X12;
	#peripheralError := #tempErrorWord.%X13;
	#synchronousError := #tempErrorWord.%X14;
	#adaptionError := #tempErrorWord.%X15;
END_FUNCTION_BLOCK

FUNCTION_BLOCK "LAxisCtrl_GetAxisWarningWord"
{ S7_Optimized_Access := 'TRUE' }
AUTHOR : 'tech.team.motioncontrol@siemens.com'
FAMILY : AxisCtrl
VERSION : 1.0
   VAR_INPUT 
      axis {InstructionName := 'TO_SpeedAxis'; LibVersion := '6.0'} : TO_SpeedAxis;
   END_VAR

   VAR_OUTPUT 
      systemWarning { ExternalWritable := 'False'; S7_HiddenAssignment := 'HideIfNoParamAssigned'} : Bool;
      configWarning { ExternalWritable := 'False'; S7_HiddenAssignment := 'HideIfNoParamAssigned'} : Bool;
      userWarning { ExternalWritable := 'False'; S7_HiddenAssignment := 'HideIfNoParamAssigned'} : Bool;
      commandNotAccepted { ExternalWritable := 'False'; S7_HiddenAssignment := 'HideIfNoParamAssigned'} : Bool;
      driveWarning { ExternalWritable := 'False'; S7_HiddenAssignment := 'HideIfNoParamAssigned'} : Bool;
      sensorWarning { ExternalWritable := 'False'; S7_HiddenAssignment := 'HideIfNoParamAssigned'} : Bool;
      dynamicError { ExternalWritable := 'False'; S7_HiddenAssignment := 'HideIfNoParamAssigned'} : Bool;
      communicationWarning { ExternalWritable := 'False'; S7_HiddenAssignment := 'HideIfNoParamAssigned'} : Bool;
      swLimitMin { ExternalWritable := 'False'; S7_HiddenAssignment := 'HideIfNoParamAssigned'} : Bool;
      swLimitMax { ExternalWritable := 'False'; S7_HiddenAssignment := 'HideIfNoParamAssigned'} : Bool;
      homingWarning { ExternalWritable := 'False'; S7_HiddenAssignment := 'HideIfNoParamAssigned'} : Bool;
      followingErrorWarning { ExternalWritable := 'False'; S7_HiddenAssignment := 'HideIfNoParamAssigned'} : Bool;
      positioningWarning { ExternalWritable := 'False'; S7_HiddenAssignment := 'HideIfNoParamAssigned'} : Bool;
      peripheralWarning { ExternalWritable := 'False'; S7_HiddenAssignment := 'HideIfNoParamAssigned'} : Bool;
      synchronousWarning { ExternalWritable := 'False'; S7_HiddenAssignment := 'HideIfNoParamAssigned'} : Bool;
      adaptionWarning { ExternalWritable := 'False'; S7_HiddenAssignment := 'HideIfNoParamAssigned'} : Bool;
   END_VAR

   VAR_TEMP 
      tempWarningWord : DWord;
   END_VAR


BEGIN
	//==========================================================================================
	// SIEMENS AG
	// (c)Copyright 2017 All Rights Reserved
	//------------------------------------------------------------------------------------------
	// Library: LAxisCtrl
	// Tested with: S7-1515T-2 PN
	// Engineering: TIA Portal V15
	// Restrictions: ---
	// Requirements: S7-1500/S7-1500T FW 2.5
	// Functionality: The FB is splitting the warning word of an axis into bits.
	// Support: tech.team.motioncontrol@siemens.com
	// Note: Parameter comments are only available in language 'English (United States)'
	//------------------------------------------------------------------------------------------
	// Change log table:
	// Version    Date          Expert in charge    Changes applied
	// 01.00.01   04.10.2016    AL                  First released version
	// 01.00.02   29.03.2017    AL                  Added support information
	//===========================================================================================
	
	//----------------------------------------------------------------------------------------------
	// Read warningword
	//----------------------------------------------------------------------------------------------
	#tempWarningWord := #axis.WarningWord;
	
	//----------------------------------------------------------------------------------------------
	// Write outputs
	//----------------------------------------------------------------------------------------------
	#systemWarning := #tempWarningWord.%X0;
	#configWarning := #tempWarningWord.%X1;
	#userWarning := #tempWarningWord.%X2;
	#commandNotAccepted := #tempWarningWord.%X3;
	#driveWarning := #tempWarningWord.%X4;
	#sensorWarning := #tempWarningWord.%X5;
	#dynamicError := #tempWarningWord.%X6;
	#communicationWarning := #tempWarningWord.%X7;
	#swLimitMin := #tempWarningWord.%X8;
	#swLimitMax := #tempWarningWord.%X9;
	#homingWarning := #tempWarningWord.%X10;
	#followingErrorWarning := #tempWarningWord.%X11;
	#positioningWarning := #tempWarningWord.%X12;
	#peripheralWarning := #tempWarningWord.%X13;
	#synchronousWarning := #tempWarningWord.%X14;
	#adaptionWarning := #tempWarningWord.%X15;
END_FUNCTION_BLOCK

DATA_BLOCK "CONTROL_ON_FB_IDB"   // DB30230
// stored: AssignedProDiagFB GENERAL_PD, AutoNumber false, InstanceOfName CONTROL_ON_OFF_PD_FB, InstanceOfType FB
"CONTROL_ON_OFF_PD_FB"
   // VAR_INPUT
   //    PLANT_IDENTIFIER { ExternalAccessible := 'False'; ExternalVisible := 'False'; ExternalWritable := 'False'} : WString[24];
   //    ENABLE_CONTROL_ON { ExternalAccessible := 'False'; ExternalVisible := 'False'; ExternalWritable := 'False'} : Bool;
   //    PUSHBUTTON_ON { ExternalAccessible := 'False'; ExternalVisible := 'False'; ExternalWritable := 'False'} : Bool;
   //    PUSHBUTTON_OFF { ExternalAccessible := 'False'; ExternalVisible := 'False'; ExternalWritable := 'False'} : Bool;
   //    CONTACTOR_FEEDBACK { ExternalAccessible := 'False'; ExternalVisible := 'False'; ExternalWritable := 'False'} : Bool;
   //    RESET { ExternalAccessible := 'False'; ExternalVisible := 'False'; ExternalWritable := 'False'} : Bool;
   //    TIME_FEEDBACK_ON { ExternalAccessible := 'False'; ExternalVisible := 'False'; ExternalWritable := 'False'} : Time;
   //    TIME_DELAY_1 { ExternalAccessible := 'False'; ExternalVisible := 'False'; ExternalWritable := 'False'} : Time;
   //    TIME_DELAY_2 { ExternalAccessible := 'False'; ExternalVisible := 'False'; ExternalWritable := 'False'} : Time;
   //    "GLOBAL_CLOCK&SYSTEM" { ExternalAccessible := 'False'; ExternalVisible := 'False'; ExternalWritable := 'False'} : "GLOBAL_CLOCK&SYSTEM_MEMORY_UDT";
   // END_VAR
   // VAR_OUTPUT
   //    GENERAL_ALARM { ExternalAccessible := 'False'; ExternalVisible := 'False'; ExternalWritable := 'False'} : Bool;
   //    CONTACTER_ON { ExternalAccessible := 'False'; ExternalVisible := 'False'; ExternalWritable := 'False'} : Bool;
   //    CONTROL_ON { ExternalAccessible := 'False'; ExternalVisible := 'False'; ExternalWritable := 'False'} : Bool;
   //    CONTROL_ON_DELAYED_1 { ExternalAccessible := 'False'; ExternalVisible := 'False'; ExternalWritable := 'False'} : Bool;
   //    CONTROL_ON_DELAYED_2 { ExternalAccessible := 'False'; ExternalVisible := 'False'; ExternalWritable := 'False'} : Bool;
   //    EXTENDED_PULSE_PLC_ON { ExternalAccessible := 'False'; ExternalVisible := 'False'; ExternalWritable := 'False'} : Bool;
   //    CONTROL_ON_DISPLAY { ExternalAccessible := 'False'; ExternalVisible := 'False'; ExternalWritable := 'False'} : Bool;
   //    CONTROL_OFF_DISPLAY { ExternalAccessible := 'False'; ExternalVisible := 'False'; ExternalWritable := 'False'} : Bool;
   // END_VAR
   // VAR
   //    HMI_IN : Byte;
   //    HMI_ON_OFF_Header : Byte;
   //    HMI_OFF : Byte;
   //    HMI_ON : Bool;
   //    HMI_Req_OFF : Bool;
   //    Instruction { ExternalAccessible := 'False'; ExternalVisible := 'False'; ExternalWritable := 'False'} : Struct
   //       Timer_Feedback_On { S7_SetPoint := 'True'} : IEC_TIMER;
   //       Timer_Control_ON_delay_1 { S7_SetPoint := 'True'} : IEC_TIMER;
   //       Timer_Control_ON_delay_2 { S7_SetPoint := 'True'} : IEC_TIMER;
   //       Timer_Control_ON_display { S7_SetPoint := 'True'} : IEC_TIMER;
   //       PLC_delay_ON { S7_SetPoint := 'True'} : IEC_TIMER;
   //       Extended_PLC_ON { S7_SetPoint := 'True'} : IEC_TIMER;
   //    END_STRUCT;
   //    Alarm { ExternalAccessible := 'False'; ExternalVisible := 'False'; ExternalWritable := 'False'} : Struct
   //       T_FeedBack_ON : Bool;
   //       FeedBack_Lost_no_cmd : Bool;
   //       Enable_missing : Bool;
   //       Spare_3 : Bool;
   //       Spare_4 : Bool;
   //       Spare_5 : Bool;
   //       Spare_6 : Bool;
   //       Spare_7 : Bool;
   //       Spare_8 : Bool;
   //       Spare_9 : Bool;
   //       Spare_10 : Bool;
   //       Spare_11 : Bool;
   //       Spare_12 : Bool;
   //       Spare_13 : Bool;
   //       Spare_14 : Bool;
   //       Spare_15 : Bool;
   //    END_STRUCT;
   //    PE { ExternalAccessible := 'False'; ExternalVisible := 'False'; ExternalWritable := 'False'} : Struct
   //       AlarmReset : Bool;
   //       ControlON : Bool;
   //       ControlOFF : Bool;
   //       ReqOFF : Bool;
   //    END_STRUCT;
   //    PP { ExternalAccessible := 'False'; ExternalVisible := 'False'; ExternalWritable := 'False'} : Struct
   //       AlarmReset : Bool;
   //       ControlON : Bool;
   //       ControlOFF : Bool;
   //       ReqOFF : Bool;
   //    END_STRUCT;
   //    NE { ExternalAccessible := 'False'; ExternalVisible := 'False'; ExternalWritable := 'False'} : Struct
   //       Feedback_On : Bool;
   //       ReqOFF : Bool;
   //       ControlOFF : Bool;
   //    END_STRUCT;
   //    NP { ExternalAccessible := 'False'; ExternalVisible := 'False'; ExternalWritable := 'False'} : Struct
   //       Feedback_On : Bool;
   //       ReqOFF : Bool;
   //       ControlOFF : Bool;
   //    END_STRUCT;
   //    AX { ExternalAccessible := 'False'; ExternalVisible := 'False'; ExternalWritable := 'False'} : Struct
   //       FirstCycle : Bool;
   //       ControlOFF_Req : Bool;
   //       ControlOFF_active : Bool;
   //       ContactorON : Bool;
   //       General_Alarm : Bool;
   //       Control_ON_delayed_1 : Bool;
   //       Control_ON_delayed_2 : Bool;
   //       Control_ON : Bool;
   //       Extended_PLC_ON : Bool;
   //       Control_ON_display : Bool;
   //    END_STRUCT;
   //    Alarm_No_PD { ExternalAccessible := 'False'; ExternalVisible := 'False'; ExternalWritable := 'False'} : UInt;
   //    GLOBAL_GENERAL_AlarmTextList_Item { ExternalAccessible := 'False'; ExternalVisible := 'False'; ExternalWritable := 'False'} : USInt;
   // END_VAR
BEGIN
END_DATA_BLOCK

DATA_BLOCK "GLOBAL_INFO_FB_IDB"   // DB30231
AUTHOR : Tesla
FAMILY : Base
VERSION : 1.0
// stored: AutoNumber false, InstanceOfName GLOBAL_INFO_FB, InstanceOfType FB
"GLOBAL_INFO_FB"
   // VAR_INPUT
   //    NO_OPERATION_MODE { ExternalAccessible := 'False'; ExternalVisible := 'False'; ExternalWritable := 'False'} : Int;
   //    NO_HMI_PANEL { ExternalAccessible := 'False'; ExternalVisible := 'False'; ExternalWritable := 'False'} : Int;
   //    CLOCK_MEMORY { ExternalAccessible := 'False'; ExternalVisible := 'False'; ExternalWritable := 'False'} : Byte;
   //    SYSTEM_MEMORY { ExternalAccessible := 'False'; ExternalVisible := 'False'; ExternalWritable := 'False'} : Byte;
   //    RTG1SYSINFO { ExternalAccessible := 'False'; ExternalVisible := 'False'; ExternalWritable := 'False'} : F_SYSINFO;
   //    LADDR : HW_IO;
   // END_VAR
   // VAR_OUTPUT
   //    "ALWAYS=TRUE" { ExternalAccessible := 'False'; ExternalVisible := 'False'; ExternalWritable := 'False'} : Bool;
   //    "ALWAYS=FALSE" { ExternalAccessible := 'False'; ExternalVisible := 'False'; ExternalWritable := 'False'} : Bool;
   //    FIRST_CYCLE { ExternalAccessible := 'False'; ExternalVisible := 'False'; ExternalWritable := 'False'} : Bool;
   // END_VAR
   // VAR_IN_OUT
   //    INIT_HMI_OPMODE : "INIT_HMI_OPMODE_UDT";
   // END_VAR
   // VAR
   //    HMI_GLOBAL { S7_SetPoint := 'True'} : "GLOBAL_STRUCT_UDT";
   //    HMI_ClockMemory : Byte;
   // END_VAR
BEGIN
END_DATA_BLOCK

DATA_BLOCK "IF_HMI_FB_IDB"   // DB30222
// stored: AutoNumber false, InstanceOfName IF_HMI_FB, InstanceOfType FB
"IF_HMI_FB"
   // VAR_INPUT
   //    INIT_HMI_OPMODE { ExternalAccessible := 'False'; ExternalVisible := 'False'; ExternalWritable := 'False'} : "INIT_HMI_OPMODE_UDT";
   //    CLOCK_SYSTEM_INFO : "GLOBAL_CLOCK&SYSTEM_MEMORY_UDT";
   // END_VAR
   // VAR_IN_OUT
   //    OPERATOR_PROMPT_IF : "OPERATOR_PROMPT_UDT";
   // END_VAR
   // VAR
   //    "IF" { S7_SetPoint := 'True'} : "IF_HMI_UDT";
   //    "RT_INFO.INFO" { ExternalAccessible := 'False'; ExternalVisible := 'False'; ExternalWritable := 'False'} : LTime;
   //    "RT_INFO.RET_VAL" { ExternalAccessible := 'False'; ExternalVisible := 'False'; ExternalWritable := 'False'} : Word;
   //    CycleConvert { ExternalAccessible := 'False'; ExternalVisible := 'False'; ExternalWritable := 'False'} : Int;
   //    LimitValue { ExternalAccessible := 'False'; ExternalVisible := 'False'; ExternalWritable := 'False'} : Int;
   // END_VAR
BEGIN
END_DATA_BLOCK

DATA_BLOCK "OPMODE01_IDB"   // DB105
// stored: AssignedProDiagFB OPMODE01_PD, InstanceOfName COND_PD_FB, InstanceOfType FB
"COND_PD_FB"
   // VAR_INPUT
   //    PD_TEXT { ExternalAccessible := 'False'; ExternalVisible := 'False'; ExternalWritable := 'False'} : WString[24];
   //    COND_NUMBER { ExternalAccessible := 'False'; ExternalVisible := 'False'; ExternalWritable := 'False'} : Int;
   //    COND_LOGIC { ExternalAccessible := 'False'; ExternalVisible := 'False'; ExternalWritable := 'False'} : Bool;
   //    CODE_VIEW_ENABLE { ExternalAccessible := 'False'; ExternalVisible := 'False'; ExternalWritable := 'False'} : Bool;
   // END_VAR
   // VAR_OUTPUT
   //    COND_OK { ExternalAccessible := 'False'; ExternalVisible := 'False'; ExternalWritable := 'False'} : Bool;
   // END_VAR
   // VAR_IN_OUT
   //    "IF" : "COND_PD_UDT";
   // END_VAR
   // VAR
   //    Code_View_Enabled { ExternalAccessible := 'False'; ExternalVisible := 'False'; ExternalWritable := 'False'} : Bool;
   // END_VAR
BEGIN
END_DATA_BLOCK

DATA_BLOCK "OPMODE01_OPEN_DOOR_IDB"   // DB88
// stored: AssignedProDiagFB OPMODE01_PD, InstanceOfName COND_PD_FB, InstanceOfType FB
"COND_PD_FB"
   // VAR_INPUT
   //    PD_TEXT { ExternalAccessible := 'False'; ExternalVisible := 'False'; ExternalWritable := 'False'} : WString[24];
   //    COND_NUMBER { ExternalAccessible := 'False'; ExternalVisible := 'False'; ExternalWritable := 'False'} : Int;
   //    COND_LOGIC { ExternalAccessible := 'False'; ExternalVisible := 'False'; ExternalWritable := 'False'} : Bool;
   //    CODE_VIEW_ENABLE { ExternalAccessible := 'False'; ExternalVisible := 'False'; ExternalWritable := 'False'} : Bool;
   // END_VAR
   // VAR_OUTPUT
   //    COND_OK { ExternalAccessible := 'False'; ExternalVisible := 'False'; ExternalWritable := 'False'} : Bool;
   // END_VAR
   // VAR_IN_OUT
   //    "IF" : "COND_PD_UDT";
   // END_VAR
   // VAR
   //    Code_View_Enabled { ExternalAccessible := 'False'; ExternalVisible := 'False'; ExternalWritable := 'False'} : Bool;
   // END_VAR
BEGIN
END_DATA_BLOCK

DATA_BLOCK "S7通信读写_1200"   // DB5
// stored: InstanceOfName S7通信读写, InstanceOfType FB
"S7通信读写"
BEGIN
END_DATA_BLOCK

DATA_BLOCK "S7通信读写_G2"   // DB3
// stored: InstanceOfName S7通信读写, InstanceOfType FB
"S7通信读写"
BEGIN
END_DATA_BLOCK

DATA_BLOCK "FB_IO_Map_Disp_IDB"   // DB101
// stored: AutoNumber false, InstanceOfName FB_IO_Map_Disp, InstanceOfType FB
"FB_IO_Map_Disp"
BEGIN
END_DATA_BLOCK

DATA_BLOCK "放卷伺服S120"   // DB1, Motion_DB
// stored: InstanceOfName TO_PositioningAxis, OfSystemLibElement TO_PositioningAxis, OfSystemLibVersion 6.0
TO_PositioningAxis   // technology object, version 6.0
   // // inherited from TO_SpeedAxis
   // // inherited from TO_Axis
   // // inherited from TO_Object
   // VAR
   //    Actor : TO_Struct_Actor;
   //    Simulation : TO_Struct_AxisSimulation;
   // END_VAR
   // VAR
   //    Position { ExternalWritable := 'False'} : LReal;
   //    ActualPosition { ExternalWritable := 'False'} : LReal;
   //    ActualVelocity { ExternalWritable := 'False'} : LReal;
   //    ActualAcceleration { ExternalWritable := 'False'} : LReal;
   //    OperativeSensor { ExternalWritable := 'False'} : UDInt;
   //    ModuloCycle { ExternalWritable := 'False'} : DInt;
   //    ActualModuloCycle { ExternalWritable := 'False'} : DInt;
   //    Clamping { S7_SetPoint := 'True'} : TO_Struct_Clamping;
   //    Sensor { S7_SetPoint := 'True'} : Array[1..4] of TO_Struct_Sensor;
   //    Extrapolation { S7_SetPoint := 'True'} : TO_Struct_Extrapolation;
   //    Mechanics { S7_SetPoint := 'True'} : TO_Struct_Mechanics;
   //    Properties { ExternalWritable := 'False'; S7_SetPoint := 'True'} : TO_Struct_Properties;
   //    Modulo { S7_SetPoint := 'True'} : TO_Struct_Modulo;
   //    PositionLimits_SW { S7_SetPoint := 'True'} : TO_Struct_PositionLimitsSW;
   //    PositionLimits_HW { S7_SetPoint := 'True'} : TO_Struct_PositionLimitsHW;
   //    Homing { S7_SetPoint := 'True'} : TO_Struct_Homing;
   //    PositionControl { S7_SetPoint := 'True'} : TO_Struct_PositionControl;
   //    DynamicAxisModel { S7_SetPoint := 'True'} : TO_Struct_DynamicAxisModel;
   //    FollowingError { S7_SetPoint := 'True'} : TO_Struct_FollowingError;
   //    CrossPlcSynchronousOperation { S7_SetPoint := 'True'} : TO_Struct_CrossPlcSynchronousOperation;
   //    PositioningMonitoring { S7_SetPoint := 'True'} : TO_Struct_PositioningMonitoring;
   //    StandstillSignal { S7_SetPoint := 'True'} : TO_Struct_StandstillSignal;
   //    StatusPositioning { ExternalWritable := 'False'; S7_SetPoint := 'True'} : TO_Struct_StatusPositioning;
   //    StatusServo { ExternalWritable := 'False'; S7_SetPoint := 'True'} : TO_Struct_StatusServo;
   //    StatusProvidedLeadingValue { ExternalWritable := 'False'; S7_SetPoint := 'True'} : TO_Struct_StatusProvidedLeadingValue;
   //    StatusSensor { ExternalWritable := 'False'; S7_SetPoint := 'True'} : Array[1..4] of TO_Struct_StatusSensor;
   //    StatusExtrapolation { ExternalWritable := 'False'; S7_SetPoint := 'True'} : TO_Struct_StatusExtrapolation;
   //    StatusKinematicsMotion { ExternalWritable := 'False'; S7_SetPoint := 'True'} : TO_Struct_StatusKinematicsMotion;
   // END_VAR
BEGIN
   Actor.DataAdaption := 1;
   Actor.Interface.AddressIn.RID := 16#208071a;
   Actor.Interface.AddressIn.AREA := 16#81;
   Actor.Interface.AddressIn.OFFSET := 1032;
   Actor.Interface.AddressOut.RID := 16#208071b;
   Actor.Interface.AddressOut.AREA := 16#82;
   Actor.Interface.AddressOut.OFFSET := 1056;
   Simulation.Mode := 1;
   Sensor[1].DataAdaption := 1;
   Sensor[1].Interface.AddressIn.RID := 16#208071a;
   Sensor[1].Interface.AddressIn.AREA := 16#81;
   Sensor[1].Interface.AddressIn.OFFSET := 1032;
   Sensor[1].Interface.AddressOut.RID := 16#208071b;
   Sensor[1].Interface.AddressOut.AREA := 16#82;
   Sensor[1].Interface.AddressOut.OFFSET := 1056;
   Sensor[1].ActiveHoming.Mode := 2;
   Sensor[1].ActiveHoming.DigitalInputAddress.RID := 16#2000001;
   Sensor[1].ActiveHoming.DigitalInputAddress.AREA := 16#81;
   Sensor[1].ActiveHoming.DigitalInputAddress.OFFSET := 2;
   PositionLimits_HW.Active := true;
   PositionLimits_HW.MinSwitchAddress.RID := 16#2000001;
   PositionLimits_HW.MinSwitchAddress.AREA := 16#81;
   PositionLimits_HW.MinSwitchAddress.OFFSET := 1;
   PositionLimits_HW.MaxSwitchAddress.RID := 16#2000001;
   PositionLimits_HW.MaxSwitchAddress.AREA := 16#81;
   Homing.AutoReversal := true;
   PositionControl.EnableDSC := true;
   _Sensor[1].ActiveHoming.DigitalInputAddress := s120原点信号;
   _PositionLimits_HW.MinSwitchAddress := s120负限位;
   _PositionLimits_HW.MaxSwitchAddress := S120正限位;
   _Actor.Interface.Telegram := 5;
   _Sensor[1].Interface.Telegram := 5;
END_DATA_BLOCK

